	// Statemachine
	eStep					:E_ModbusRtuMaster_State;	// State
	eStepPrevious			:E_ModbusRtuMaster_State;	// State from previous scan
	eStatePrevious			:E_ModbusRtuMaster_State;	// Previous state
	nStepSecCount			:UDINT;						// Counts number of seconds without state transitions
	wStateSecOld			:WORD;						// Seconds value from NtTime from previous scan	
	eStepEntry				:BOOL;						// True in one scan when a new state is entered
	arrStateLog				:ARRAY[0..19] OF ST_ModbusRtuMaster_StateLogEntry; // Log that contains the last xx states
	
	// Modbus master
	fbModBusMaster			:ModbusRtuMaster_KL6x22B;	// Modbus master functions
	bReadExe				:BOOL;						// On rising edge reading is started
	bReadBusy				:BOOL;						// True while modbus master reads register on unit
	bReadError				:BOOL;						// True if read error occured
	eReadErrorID			:MODBUS_ERRORS;				// Modbus error ID
	nReadNoOfBytes			:UINT;						// Nunber of bytes read in read cycle

	// Units
	nUnitActive				:INT;						// Active unit in cyclic read
	nParamActive			:INT;						// Active parameter in cyclic read
END_VAR
VAR CONSTANT
	cNoOfUnitsMax			:INT:= 20;					// Maximum number of units for modbus master
END_VAR


// Initialization	
IF bInit THEN	
	bInit := FALSE;
END_IF

// Wait for reset
IF bCmdReset THEN
	bCmdReset := FALSE;
	bError := FALSE;
	nErrorUnit := 0;
	bReadExe := FALSE;
	eStep := E_ModbusRtuMaster_State.eIdle;	
END_IF

// Update fb for modbus communication
IF eStep >= E_ModbusRtuMaster_State.eReadPre AND eStep <= E_ModbusRtuMaster_State.eReadPost THEN
	fbModbusMaster.ReadRegs(
		UnitID:= pUnit^[nUnitActive].nAddr, 
		Quantity:= pUnit^[nUnitActive].aParam[nParamActive].nQuantity, 
		MBAddr:= (pUnit^[nUnitActive].aParam[nParamActive].nMemAddr*10)-1, 
		cbLength:= pUnit^[nUnitActive].aParam[nParamActive].nQuantity*2, 
		pMemoryAddr:= ADR(pUnit^[nUnitActive].aParam[nParamActive].aDataStorage), 
		Execute:= bReadExe, 
		Timeout:= T#2S, 
		BUSY=> bReadBusy, 
		Error=> bReadError, 
		ErrorId=> eReadErrorID, 
		cbRead=> nReadNoOfBytes);	
END_IF

	
// State machine
//----------------------------------------
// Check for new state entry
IF eStep <> eStepPrevious THEN
	// New state, Set entry flag
	eStepEntry := TRUE;
	eStatePrevious := eStepPrevious;
ELSE
	// Same state as last scan, remove entry flag
	eStepEntry := FALSE;
END_IF
// Update state log
A_StateLog();
// Reset "old" state to present value
eStepPrevious := eStep;
	

CASE eStep OF
E_ModbusRtuMaster_State.eReset:
	eStep := E_ModbusRtuMaster_State.eIdle;	


E_ModbusRtuMaster_State.eIdle:
	// Entry
	IF eStepEntry THEN
		A_ResetAllCmd();
		bBusy 	:= FALSE;
		bError	:= FALSE;
		bReadExe := FALSE;
	END_IF
	// Wait for command
	IF bCmdCyclicRead THEN
		bBusy	 := TRUE;
		bReadExe := FALSE;
		bCmdCyclicRead := FALSE;
		nUnitActive := 1;
		nParamActive := 1;
		eStep := E_ModbusRtuMaster_State.eReadPre;
	END_IF
		
	
E_ModbusRtuMaster_State.eReadPre:
	// Send request for reading of hold register
	bReadExe := TRUE;
	//IF bReadBusy THEN
		eStep := E_ModbusRtuMaster_State.eReadPost;
	//END_IF	 
	
	
E_ModbusRtuMaster_State.eReadPost:
	// Wait for answer back
	IF NOT bReadBusy THEN
		IF NOT bReadError THEN
			// Successfull read
			nReadCount := nReadCount + 1;
			// Convert return data to value
			IF pUnit^[nUnitActive].aParam[nParamActive].eDataType = E_Modbus_DataType.eInt16 THEN
				nValueTempInt16 := FUN_ConvTwoByteToInt16(
									nValue1:= pUnit^[nUnitActive].aParam[nParamActive].aDataStorage[1],
									nValue2:= pUnit^[nUnitActive].aParam[nParamActive].aDataStorage[2]);
				pUnit^[nUnitActive].aParam[nParamActive].aDataValue := INT_TO_REAL(nValueTempInt16) * pUnit^[nUnitActive].aParam[nParamActive].fConvFactor;				
			ELSIF pUnit^[nUnitActive].aParam[nParamActive].eDataType = E_Modbus_DataType.eInt32 THEN
				nValueTempInt32 := FUN_ConvFourByteToInt32(
									nValue1:= pUnit^[nUnitActive].aParam[nParamActive].aDataStorage[3],
									nValue2:= pUnit^[nUnitActive].aParam[nParamActive].aDataStorage[4],
									nValue3:= pUnit^[nUnitActive].aParam[nParamActive].aDataStorage[1],
									nValue4:= pUnit^[nUnitActive].aParam[nParamActive].aDataStorage[2]);
				pUnit^[nUnitActive].aParam[nParamActive].aDataValue := DINT_TO_REAL(nValueTempInt32) * pUnit^[nUnitActive].aParam[nParamActive].fConvFactor; 
			END_IF
			// Determine next step
			IF NOT bCmdStop THEN
				// Update setting to next parameter (and unit if this was the last parameter)
				nParamActive := nParamActive + 1;
				IF nParamActive > nNoOfParam THEN
					// All parameters read from unit. Change to next unit
					nParamActive := 1;
					IF nUnitActive >= nNoOfUnits THEN
						// Loop back to first unit in array
						nUnitActive := 1;
					ELSE
						// Take next unit in array
						nUnitActive := nUnitActive + 1;
					END_IF		
				END_IF
				// Go back and start reading the next parameter
				bReadExe := FALSE;
				eStep := E_ModbusRtuMaster_State.eReadPre;
			ELSE
				// Stop cyclic reading of hold registers
				eStep := E_ModbusRtuMaster_State.eIdle;
			END_IF
		ELSE
			// Error occured
			eStep := E_ModbusRtuMaster_State.eError;	
		END_IF	
	END_IF

	
E_ModbusRtuMaster_State.eError:
	// Entry
	IF eStepEntry THEN
		A_ResetAllCmd();
		bBusy := FALSE;
		IF nErrorUnit = 0 THEN
			bError := TRUE;	 
			nErrorUnit := nUnitActive;
		END_IF
	END_IF
	
	// Go back and try next unit
	IF nUnitActive >= nNoOfUnits THEN
		// Loop back to first unit in array
		nUnitActive := 1;
	ELSE
		// Take next unit in array
		nUnitActive := nUnitActive + 1;
	END_IF
	// Go back and start reading the next parameter
	bReadExe := FALSE;
	eStep := E_ModbusRtuMaster_State.eReadPre;
	
	(*
	// Wait for reset
	IF bCmdReset THEN
		bCmdReset := FALSE;
		eStep := E_ModbusRtuMaster_State.eIdle;	
	END_IF
	*)
END_CASE

ACTION A_ResetAllCmd:
// Reset all commands
bCmdCyclicRead := FALSE;
bCmdStop  := FALSE;
bCmdReset := FALSE;
END_ACTION

ACTION A_StateLog:
// Action: State log
//---------------------------------------------------------------
// The code below implements a simple state log in RAM. The purpose of the log
// is to give the developer a state history when debugging.

// Seconds counter
//-----------------------------------------------
IF wStateSecOld <> GVL_System.stNtTime.wSecond THEN
	// New second => Update counter
	IF nStepSecCount >= 4294967294 THEN
		nStepSecCount := 0;
	END_IF
	nStepSecCount := nStepSecCount + 1;
END_IF  
wStateSecOld := GVL_System.stNtTime.wSecond;

// Update time in active state
//-----------------------------------------------
arrStateLog[0].iSecCount := nStepSecCount;

// Update Stringer state log
//-----------------------------------------------
IF 	(eStep <> eStepPrevious) THEN
	// New state transition has occured => make new entry in the state log
	// Start with shift in log (FIFO)
	MEMMOVE(
		destAddr:= ADR(arrStateLog[1]), 
		srcAddr:= ADR(arrStateLog[0]), 
		n:= (SIZEOF(arrStateLog) - SIZEOF(arrStateLog[0]))); 
		
	// Add new entry to start of log
	arrStateLog[0].eStep 		:= eStep; 
	arrStateLog[0].sTimeEntry 	:= FUN_GetTimestamp(GVL_System.stNtTime);
	arrStateLog[0].iSecCount 	:= 0;
	
	// Reset seconds counter
	nStepSecCount := 0;
END_IF
END_ACTION

METHOD M_CmdCyclicRead : BOOL
VAR_INPUT
END_VAR

// Check if it is a valid command
IF eStep = E_ModbusRtuMaster_State.eIdle THEN
	// Valid command
	bCmdCyclicRead := TRUE;
END_IF

// Return result for acceptance of command
IF bCmdCyclicRead THEN
	M_CmdCyclicRead := TRUE;
ELSE
	M_CmdCyclicRead := FALSE;
END_IF
END_METHOD

METHOD M_CmdReset : BOOL
VAR_INPUT
END_VAR

// Check if it is a valid command
IF eStep = E_ModbusRtuMaster_State.eError THEN
	// Valid command
	bCmdReset := TRUE;
END_IF

// Return result for acceptance of command
IF bCmdReset THEN
	M_CmdReset := TRUE;
ELSE
	M_CmdReset := FALSE;
END_IF
END_METHOD

METHOD M_CmdStop : BOOL
VAR_INPUT
END_VAR

// Check if it is a valid command
IF eStep > E_ModbusRtuMaster_State.eIdle AND eStep < E_ModbusRtuMaster_State.eError THEN
	// Valid command
	bCmdStop := TRUE;
END_IF

// Return result for acceptance of command
IF bCmdStop THEN
	M_CmdStop := TRUE;
ELSE
	M_CmdStop := FALSE;
END_IF
END_METHOD

END_FUNCTION_BLOCK

// ---- POUs/00_BuildingBlocks/StringFunctions/FUN_GetTimestamp.TcPOU
FUNCTION FUN_GetTimestamp : STRING
VAR_INPUT
	stNtTime		:TIMESTRUCT;
END_VAR
VAR
	sTimestamp		:STRING;
END_VAR

// Add data
sTimeStamp := FUN_GetDate(stNtTime);

// Add time
sTimestamp := CONCAT(sTimeStamp, ' ');
sTimestamp := CONCAT(sTimeStamp, FUN_GetTime(stNtTime));

// Return time stamp
FUN_GetTimestamp := sTimestamp;

END_FUNCTION

// ---- POUs/00_BuildingBlocks/StringFunctions/FUN_GetDate.TcPOU
FUNCTION FUN_GetDate : STRING
VAR_INPUT
	stNtTime		:TIMESTRUCT;
END_VAR
VAR
	sDate			:STRING;
END_VAR

// Initialize string
sDate := '';

// Add year to string
sDate := UINT_TO_STRING(stNtTime.wYear);
sDate := CONCAT(sDate,'-');

// Add month to string
IF stNtTime.wMonth < 10 THEN
	sDate := CONCAT(sDate,'0');
END_IF
sDate := CONCAT(sDate,UINT_TO_STRING(stNtTime.wMonth));
sDate := CONCAT(sDate,'-');

// Add day to string
IF stNtTime.wDay < 10 THEN
	sDate := CONCAT(sDate, '0');
END_IF
sDate := CONCAT(sDate,UINT_TO_STRING(stNtTime.wDay));

// Return result
FUN_GetDate := sDate;

END_FUNCTION

// ---- POUs/00_BuildingBlocks/StringFunctions/FUN_GetTime.TcPOU
FUNCTION FUN_GetTime : STRING
VAR_INPUT
	stNtTime		:TIMESTRUCT;
END_VAR
VAR
	sTimestamp		:STRING;
END_VAR

// Add hour to timestamp
sTimestamp := '';
IF stNtTime.wHour < 10 THEN
	sTimestamp := CONCAT(sTimestamp,CONCAT('0', UINT_TO_STRING(stNtTime.wHour)));
ELSE
	sTimestamp := CONCAT(sTimestamp,UINT_TO_STRING(stNtTime.wHour));
END_IF

// Add min to timestamp
sTimestamp := CONCAT(sTimestamp, ':');
IF stNtTime.wMinute < 10 THEN
	sTimestamp := CONCAT(sTimestamp,CONCAT('0', UINT_TO_STRING(stNtTime.wMinute)));
ELSE
	sTimestamp := CONCAT(sTimestamp,UINT_TO_STRING(stNtTime.wMinute));
END_IF
sTimestamp := CONCAT(sTimestamp, ':');

// Add sec to timestamp
IF stNtTime.wSecond < 10 THEN
	sTimestamp := CONCAT(sTimestamp,CONCAT('0', UINT_TO_STRING(stNtTime.wSecond)));
ELSE
	sTimestamp := CONCAT(sTimestamp,UINT_TO_STRING(stNtTime.wSecond));
END_IF

// Return time
FUN_GetTime := sTimestamp;

END_FUNCTION

// ---- POUs/00_BuildingBlocks/Modbus/FB_ModbusRtuMaster_20220719_1144.TcPOU
// FB_ModbusMaster
//------------------------------------------------------ 
// This FB must be called in a 2 ms task and in every scan
// Test with Danfoss FC301 shows that up to approximately 46 registers can be read pr. sec.
// Test was done with baud 115200. 
FUNCTION_BLOCK FB_ModbusRtuMaster_20220719_1144
VAR_INPUT
	pUnit					:POINTER TO ARRAY[1..cNoOfUnitsMax] OF ST_Modbus_Unit;
	nNoOfUnits				:INT;			// Number of modbus units. Maximum value is 20.					
	nNoOfParam				:INT;			// Number of modbus parameters to be read from unit. Maximum value is determined by ST_Modbus_Unit. 
END_VAR
VAR_OUTPUT
	bBusy					:BOOL;			// True while command is beeing executed
	bError					:BOOL;			// True if an error occured during execution of a command
END_VAR
VAR
	// Commands
	bCmdCyclicRead			:BOOL;			// Command for cyclic reading of parameter registers
	bCmdStop				:BOOL;			// Command for stop
	bCmdReset				:BOOL;			// Command for reset of active errors
	
	// General	
	bInit					:BOOL := TRUE;	// True at the start of false scan, false otherwise
	nReadCount				:INT;			// Counts the number of succesfull read operations
	nValueTempInt16			:INT;			// Value used in conversion from byte data to actual data value
	nValueTempInt32			:DINT;			// Value used in conversion from byte data to actual data value
	
	// Statemachine
	eStep					:E_ModbusRtuMaster_State;	// State
	eStepPrevious				:E_ModbusRtuMaster_State;	// State from previous scan
	eStatePrevious			:E_ModbusRtuMaster_State;	// Previous state
	nStepSecCount			:UDINT;						// Counts number of seconds without state transitions
	wStateSecOld			:WORD;						// Seconds value from NtTime from previous scan	
	eStepEntry				:BOOL;						// True in one scan when a new state is entered
	arrStateLog				:ARRAY[0..19] OF ST_ModbusRtuMaster_StateLogEntry; // Log that contains the last xx states
	
	// Modbus master
	fbModBusMaster			:ModbusRtuMaster_KL6x22B;	// Modbus master functions
	bReadExe				:BOOL;						// On rising edge reading is started
	bReadBusy				:BOOL;						// True while modbus master reads register on unit
	bReadError				:BOOL;						// True if read error occured
	eReadErrorID			:MODBUS_ERRORS;				// Modbus error ID
	nReadNoOfBytes			:UINT;						// Nunber of bytes read in read cycle

	// Units
	nUnitActive				:INT;						// Active unit in cyclic read
	nParamActive			:INT;						// Active parameter in cyclic read
END_VAR
VAR CONSTANT
	cNoOfUnitsMax			:INT:= 20;					// Maximum number of units for modbus master
END_VAR


// Initialization	
IF bInit THEN	
	bInit := FALSE;
END_IF


// Update fb for modbus communication
IF eStep >= E_ModbusRtuMaster_State.eReadPre AND eStep <= E_ModbusRtuMaster_State.eReadPost THEN
	fbModbusMaster.ReadRegs(
		UnitID:= pUnit^[nUnitActive].nAddr, 
		Quantity:= pUnit^[nUnitActive].aParam[nParamActive].nQuantity, 
		MBAddr:= (pUnit^[nUnitActive].aParam[nParamActive].nMemAddr*10)-1, 
		cbLength:= pUnit^[nUnitActive].aParam[nParamActive].nQuantity*2, 
		pMemoryAddr:= ADR(pUnit^[nUnitActive].aParam[nParamActive].aDataStorage), 
		Execute:= bReadExe, 
		Timeout:= T#2S, 
		BUSY=> bReadBusy, 
		Error=> bReadError, 
		ErrorId=> eReadErrorID, 
		cbRead=> nReadNoOfBytes);	
END_IF

	
// State machine
//----------------------------------------
// Check for new state entry
IF eStep <> eStepPrevious THEN
	// New state, Set entry flag
	eStepEntry := TRUE;
	eStatePrevious := eStepPrevious;
ELSE
	// Same state as last scan, remove entry flag
	eStepEntry := FALSE;
END_IF
// Update state log
A_StateLog();
// Reset "old" state to present value
eStepPrevious := eStep;
	

CASE eStep OF
E_ModbusRtuMaster_State.eReset:
	eStep := E_ModbusRtuMaster_State.eIdle;	


E_ModbusRtuMaster_State.eIdle:
	// Entry
	IF eStepEntry THEN
		A_ResetAllCmd();
		bBusy 	:= FALSE;
		bError	:= FALSE;
		bReadExe := FALSE;
	END_IF
	// Wait for command
	IF bCmdCyclicRead THEN
		bBusy	 := TRUE;
		bReadExe := FALSE;
		bCmdCyclicRead := FALSE;
		nUnitActive := 1;
		nParamActive := 1;
		eStep := E_ModbusRtuMaster_State.eReadPre;
	END_IF
		
	
E_ModbusRtuMaster_State.eReadPre:
	// Send request for reading of hold register
	bReadExe := TRUE;
	//IF bReadBusy THEN
		eStep := E_ModbusRtuMaster_State.eReadPost;
	//END_IF	 
	
	
E_ModbusRtuMaster_State.eReadPost:
	// Wait for answer back
	IF NOT bReadBusy THEN
		IF NOT bReadError THEN
			// Successfull read
			nReadCount := nReadCount + 1;
			// Convert return data to value
			IF pUnit^[nUnitActive].aParam[nParamActive].eDataType = E_Modbus_DataType.eInt16 THEN
				nValueTempInt16 := FUN_ConvTwoByteToInt16(
									nValue1:= pUnit^[nUnitActive].aParam[nParamActive].aDataStorage[1],
									nValue2:= pUnit^[nUnitActive].aParam[nParamActive].aDataStorage[2]);
				pUnit^[nUnitActive].aParam[nParamActive].aDataValue := INT_TO_REAL(nValueTempInt16) * pUnit^[nUnitActive].aParam[nParamActive].fConvFactor;				
			ELSIF pUnit^[nUnitActive].aParam[nParamActive].eDataType = E_Modbus_DataType.eInt32 THEN
				nValueTempInt32 := FUN_ConvFourByteToInt32(
									nValue1:= pUnit^[nUnitActive].aParam[nParamActive].aDataStorage[3],
									nValue2:= pUnit^[nUnitActive].aParam[nParamActive].aDataStorage[4],
									nValue3:= pUnit^[nUnitActive].aParam[nParamActive].aDataStorage[1],
									nValue4:= pUnit^[nUnitActive].aParam[nParamActive].aDataStorage[2]);
				pUnit^[nUnitActive].aParam[nParamActive].aDataValue := DINT_TO_REAL(nValueTempInt32) * pUnit^[nUnitActive].aParam[nParamActive].fConvFactor; 
			END_IF
			// Determine next step
			IF NOT bCmdStop THEN
				// Update setting to next parameter (and unit if this was the last parameter)
				nParamActive := nParamActive + 1;
				IF nParamActive > nNoOfParam THEN
					// All parameters read from unit. Change to next unit
					nParamActive := 1;
					IF nUnitActive >= nNoOfUnits THEN
						// Loop back to first unit in array
						nUnitActive := 1;
					ELSE
						// Take next unit in array
						nUnitActive := nUnitActive + 1;
					END_IF		
				END_IF
				// Go back and start reading the next parameter
				bReadExe := FALSE;
				eStep := E_ModbusRtuMaster_State.eReadPre;
			ELSE
				// Stop cyclic reading of hold registers
				eStep := E_ModbusRtuMaster_State.eIdle;
			END_IF
		ELSE
			// Error occured
			eStep := E_ModbusRtuMaster_State.eError;	
		END_IF	
	END_IF

	
E_ModbusRtuMaster_State.eError:
	// Entry
	IF eStepEntry THEN
		A_ResetAllCmd();
		bBusy := FALSE;
		bError := TRUE;	
	END_IF
	// Wait for reset
	IF bCmdReset THEN
		bCmdReset := FALSE;
		eStep := E_ModbusRtuMaster_State.eIdle;	
	END_IF
END_CASE

ACTION A_ResetAllCmd:
// Reset all commands
bCmdCyclicRead := FALSE;
bCmdStop  := FALSE;
bCmdReset := FALSE;
END_ACTION

ACTION A_StateLog:
// Action: State log
//---------------------------------------------------------------
// The code below implements a simple state log in RAM. The purpose of the log
// is to give the developer a state history when debugging.

// Seconds counter
//-----------------------------------------------
IF wStateSecOld <> GVL_System.stNtTime.wSecond THEN
	// New second => Update counter
	IF nStepSecCount >= 4294967294 THEN
		nStepSecCount := 0;
	END_IF
	nStepSecCount := nStepSecCount + 1;
END_IF  
wStateSecOld := GVL_System.stNtTime.wSecond;

// Update time in active state
//-----------------------------------------------
arrStateLog[0].iSecCount := nStepSecCount;

// Update Stringer state log
//-----------------------------------------------
IF 	(eStep <> eStepPrevious) THEN
	// New state transition has occured => make new entry in the state log
	// Start with shift in log (FIFO)
	MEMMOVE(
		destAddr:= ADR(arrStateLog[1]), 
		srcAddr:= ADR(arrStateLog[0]), 
		n:= (SIZEOF(arrStateLog) - SIZEOF(arrStateLog[0]))); 
		
	// Add new entry to start of log
	arrStateLog[0].eStep 		:= eStep; 
	arrStateLog[0].sTimeEntry 	:= FUN_GetTimestamp(GVL_System.stNtTime);
	arrStateLog[0].iSecCount 	:= 0;
	
	// Reset seconds counter
	nStepSecCount := 0;
END_IF
END_ACTION

METHOD M_CmdCyclicRead : BOOL
VAR_INPUT
END_VAR

// Check if it is a valid command
IF eStep = E_ModbusRtuMaster_State.eIdle THEN
	// Valid command
	bCmdCyclicRead := TRUE;
END_IF

// Return result for acceptance of command
IF bCmdCyclicRead THEN
	M_CmdCyclicRead := TRUE;
ELSE
	M_CmdCyclicRead := FALSE;
END_IF
END_METHOD

METHOD M_CmdReset : BOOL
VAR_INPUT
END_VAR

// Check if it is a valid command
IF eStep = E_ModbusRtuMaster_State.eError THEN
	// Valid command
	bCmdReset := TRUE;
END_IF

// Return result for acceptance of command
IF bCmdReset THEN
	M_CmdReset := TRUE;
ELSE
	M_CmdReset := FALSE;
END_IF
END_METHOD

METHOD M_CmdStop : BOOL
VAR_INPUT
END_VAR

// Check if it is a valid command
IF eStep > E_ModbusRtuMaster_State.eIdle AND eStep < E_ModbusRtuMaster_State.eError THEN
	// Valid command
	bCmdStop := TRUE;
END_IF

// Return result for acceptance of command
IF bCmdStop THEN
	M_CmdStop := TRUE;
ELSE
	M_CmdStop := FALSE;
END_IF
END_METHOD

END_FUNCTION_BLOCK

// ---- POUs/00_BuildingBlocks/Modbus/PRG_ModbusTest.TcPOU
PROGRAM PRG_ModbusTest
VAR
	// General	
	bInit					:BOOL := TRUE;
	nForIndex				:INT;
	
	bTestCyclicRead			:BOOL;
	bTestStop				:BOOL;
	bTestReset				:BOOL;
	
	// Modbus
	fbModbus				:FB_ModbusRtuMaster;
	fbModbusBusy			:BOOL;
	fbModbusError			:BOOL;
	
	// Frequency inverters
	aVFD					:ARRAY[1..cNoOfUnits] OF ST_Modbus_Unit; 	
END_VAR
VAR CONSTANT
	cNoOfUnits				:INT:= 2;
	cNoOfParam				:INT:= 4;
END_VAR


// Initialization
//-------------------------------------------	
IF bInit THEN	
	// VFD address 
	aVFD[1].nAddr := 2;
	aVFD[2].nAddr := 3;
	// Parameters to be read in each VFD
	FOR nForIndex := 1 TO cNoOfUnits BY 1 DO
		aVFD[nForIndex].aParam[1].nMemAddr 		:= 1610;	 				 // [W] Power (Value back is in W and not kW)
		aVFD[nForIndex].aParam[1].nQuantity 	:= 4;						 // Bytes
		aVFD[nForIndex].aParam[1].fConvFactor 	:= 10.0; 				     // Conversion index 1 => Conversion factor 10
		aVFD[nForIndex].aParam[1].eDataType 	:= E_Modbus_DataType.eInt32; // Int32
		
		aVFD[nForIndex].aParam[2].nMemAddr 		:= 1612;					// [V] Motor voltage
		aVFD[nForIndex].aParam[2].nQuantity 	:= 2;						// Bytes -> 2 bytes
		aVFD[nForIndex].aParam[2].fConvFactor 	:= 0.1; 					// Conversion index -1 => Conversion factor 0.1
		aVFD[nForIndex].aParam[2].eDataType 	:= E_Modbus_DataType.eInt16;// Int16 
		
		aVFD[nForIndex].aParam[3].nMemAddr 		:= 1613;					// [Hz] Frequency
		aVFD[nForIndex].aParam[3].nQuantity 	:= 2;						// Bytes
		aVFD[nForIndex].aParam[3].fConvFactor 	:= 0.1; 					// Conversion index -1 => Conversion factor 0.1
		aVFD[nForIndex].aParam[3].eDataType 	:= E_Modbus_DataType.eInt16;// Int16 
		
		aVFD[nForIndex].aParam[4].nMemAddr 		:= 1614;					// [A] Motor current 
		aVFD[nForIndex].aParam[4].nQuantity 	:= 4;						// Bytes
		aVFD[nForIndex].aParam[4].fConvFactor 	:= 0.01;				 	// Conversion index -2 => Conversion factor 0.01
		aVFD[nForIndex].aParam[4].eDataType 	:= E_Modbus_DataType.eInt32;// Int32
	END_FOR
	bInit := FALSE;
END_IF


// Update function block that handles modbus communication
//-------------------------------------------	
fbModbus(
	pUnit:= ADR(aVFD),
	nNoOfUnits := cNoOfUnits,
	nNoOfParam := cNoOfParam,
	bBusy => fbModbusBusy,
	bError => fbModbusError);

	
// Commands	
//-------------------------------------------		
// Test/Start cyclic read of data
IF bTestCyclicRead THEN
	fbModbus.M_CmdCyclicRead();
	bTestCyclicRead := FALSE;
END_IF

// Stop cyclic read of data
IF bTestStop THEN
	fbModbus.M_CmdStop();
	bTestStop := FALSE;
END_IF

// Reset of error
IF bTestReset THEN
	fbModbus.M_CmdReset();
	bTestReset := FALSE;
END_IF

	
// Results (Read outs)
//-------------------------------------
// VFD 1
//aVFD[1].aParam[1].aDataValue;		// [W] Power
//aVFD[1].aParam[2].aDataValue;		// [V] Motor voltage
//aVFD[1].aParam[3].aDataValue;		// [Hz] Frequency
//aVFD[1].aParam[4].aDataValue;		// [A] Motor current 

// VFD 2
//aVFD[2].aParam[1].aDataValue;		// [W] Power
//aVFD[2].aParam[2].aDataValue;		// [V] Motor voltage
//aVFD[2].aParam[3].aDataValue;		// [Hz] Frequency
//aVFD[2].aParam[4].aDataValue;		// [A] Motor current

END_PROGRAM

// ---- POUs/00_BuildingBlocks/PlcToPlcCom/FB_PlcAdsRead.TcPOU
//**************************************************************************
// FB_PlcAdsRead
// -------------------------------------------------------------------------
// This FB reads the content of a variable or struct from a remote PLC. The
// FB is usefull when data needs to be exchaged between two PLC's. The FB only
// reads the content from the other PLC, it does NOT write any variables. Hence
// the same FB will need to be implemented on other PLC, which then reads the
// commands/variables that needs to be sent.  
//
// Version
//		- V1.00.00	HHL, 21/08-2019
//**************************************************************************
FUNCTION_BLOCK FB_PlcAdsRead
VAR_INPUT
	sRemoteNetId 		:STRING; 			// Remote plc NetId
	uiRemoteAmsPort 	:UINT := 851; 		// Ams port 
	sSymbolName 		:STRING := '';		// Symbol name on remote PLC
	dwAddress 			:PVOID; 			// Variable address at local system. Name must be the same at remote
	udiLength 			:UDINT; 			// Variable length at local system. Name must be the same at remote
	tReadInterval 		:TIME := T#1S; 		// Read interval
	tReadTimeout 		:TIME := T#2S; 		// Read timeout
	
	bEnable 			:BOOL := TRUE; 		// Enable communication
	bStartRead			:BOOL;				// Force Start Read  Started
END_VAR
VAR_OUTPUT
	bLinkOk 			:BOOL; 				// Link to remote plc is ok
	bError 				:BOOL; 				// Connection error
	
	eErrorStep 			:E_PlcAdsReadStep; 	// Error step
	udiErrorId 			:UDINT; 			// Error id (ads)
END_VAR
VAR
	bEntry 				:BOOL;
	udiHandle 			:UDINT; 			// Handel
	sSymbolNameEdge 	:STRING;
	
	eStep, eStepEdge 	:E_PlcAdsReadStep;
	stHmi 				:ST_PlcAdsReadHmi; 	// Hmi data
	
	fbAdsRdWrt 			:ADSRDWRT;
	fbAdsRead 			:ADSREAD;
	fbInitRetry 		:TON; 				// Delay before retry
	fbReadInterval 		:TON; 				// Read interval timer
	osStartReadADS		:R_TRIG;			// os Start Read ADS Data
	// Force Start Read Started
	bForceStartRead: BOOL;
END_VAR

osStartReadADS(CLK:=bStartRead , Q=> );

IF osStartReadADS.Q THEN
	bForceStartRead:=TRUE;
END_IF

bEntry := eStepEdge<>eStep;
eStepEdge := eStep;


CASE eStep OF
	//-----------------------------
	// Init
	E_PlcAdsReadStep.eReset:	
		fbAdsRdWrt.WRTRD := FALSE;	
		fbAdsRead.READ := FALSE;
		
		bLinkOk := FALSE;
		bError := FALSE;
		udiErrorId := 0;
		eErrorStep := E_PlcAdsReadStep.eReset;

		eStep := E_PlcAdsReadStep.eGetRemoteInfo;	
	
	//-----------------------------
	// Get info (Index-Group/Offset)
	E_PlcAdsReadStep.eGetRemoteInfo:
		IF bEntry THEN
			fbAdsRdWrt.WRTRD := TRUE;
		END_IF
		
		IF fbAdsRdWrt.BUSY THEN
			//Read started
			eStep := E_PlcAdsReadStep.eWaitRemoteInfo;
		END_IF
	
	//-----------------------------
	// Wait for remote info
	E_PlcAdsReadStep.eWaitRemoteInfo:
		IF NOT fbAdsRdWrt.BUSY THEN
			IF NOT fbAdsRdWrt.ERR THEN
				//Get remote info ok
				sSymbolNameEdge := sSymbolName;
				IF bEnable OR bForceStartRead THEN
					eStep := E_PlcAdsReadStep.eRead;
					bForceStartRead:=FALSE;
				ELSE
					eStep := E_PlcAdsReadStep.eIdle;
				END_IF
			ELSE
				//Get remote info failed
				eErrorStep := eStep;
				udiErrorId := fbAdsRdWrt.ERRID;
				
				eStep := E_PlcAdsReadStep.eGetInfoError;
			END_IF
		END_IF
	
	//-----------------------------
	// Get info failed
	E_PlcAdsReadStep.eGetInfoError:		
		IF fbInitRetry.Q THEN
			//Retry
			eStep := E_PlcAdsReadStep.eReset;
		END_IF
		
	//-----------------------------
	// Idle
	E_PlcAdsReadStep.eIdle:		
		IF bEntry THEN
			fbAdsRead.READ := FALSE;
		END_IF
		
		IF bEnable OR bForceStartRead THEN
			IF FIND(STR1:=sSymbolName, STR2:=sSymbolNameEdge)=1 THEN
				//Symbol has'nt changed
				eStep := E_PlcAdsReadStep.eRead;
				bForceStartRead:=FALSE;
			ELSE
				eStep := E_PlcAdsReadStep.eReset;
			END_IF
			
		END_IF
	
	//-----------------------------
	// Read data
	E_PlcAdsReadStep.eRead:	
		IF bEntry THEN
			//Start read
			fbAdsRead.READ := TRUE;
			eErrorStep := E_PlcAdsReadStep.eIdle;
			udiErrorId := 0;
		END_IF
		
		IF fbAdsRead.BUSY THEN
			//Read started
			eStep := E_PlcAdsReadStep.eWaitReadDone;
		END_IF
	
	//-----------------------------
	// Wait read finished
	E_PlcAdsReadStep.eWaitReadDone:
		IF NOT fbAdsRead.BUSY THEN
			stHmi.udiS_ReadCount := stHmi.udiS_ReadCount + 1;
			IF NOT fbAdsRead.ERR THEN
				bLinkOk := TRUE;
				eStep := E_PlcAdsReadStep.eWaitBeforeNextRead;
			ELSE
				bLinkOk := FALSE;
				eStep := E_PlcAdsReadStep.eReadError;
			END_IF
		END_IF
	
	//-----------------------------	
	// Wait before next read
	E_PlcAdsReadStep.eWaitBeforeNextRead:
		IF bEntry THEN
			fbAdsRead.READ := FALSE;
		END_IF
		
		IF fbReadInterval.Q THEN
			eStep := E_PlcAdsReadStep.eRead;
		END_IF
	
	//-----------------------------
	// Read failed
	E_PlcAdsReadStep.eReadError:
		IF bEntry THEN
			//Get remote info failed
			eErrorStep := eStep;
			udiErrorId := fbAdsRead.ERRID;
			stHmi.udiS_ReadErrors := stHmi.udiS_ReadErrors + 1;
		END_IF
		
		IF fbInitRetry.Q THEN
			// Try to init
			eStep := E_PlcAdsReadStep.eReset;
		END_IF
ELSE
	eStep := E_PlcAdsReadStep.eReset;
END_CASE

//Timers
fbReadInterval(IN:=NOT fbReadInterval.Q, PT:=tReadInterval);
IF fbReadInterval.Q AND (eStep=E_PlcAdsReadStep.eRead OR eStep=E_PlcAdsReadStep.eWaitReadDone) THEN
	//Read interval error
	stHmi.udiS_ReadIntervalErrors := stHmi.udiS_ReadIntervalErrors + 1;
END_IF
fbInitRetry(IN:=eStep=E_PlcAdsReadStep.eGetInfoError OR eStep=E_PlcAdsReadStep.eReadError, PT:=T#10S);

//Init
IF stHmi.bC_Init THEN
	eStep := E_PlcAdsReadStep.eReset;
	stHmi.bC_Init := FALSE;
END_IF

//Calls
fbAdsRdWrt(
	NETID:=sRemoteNetId, 
	PORT:=uiRemoteAmsPort, 
	IDXGRP:=16#F003, //GET_SYMHANDLE_BYNAME
	IDXOFFS:= 16#0000, 
	WRITELEN:= SIZEOF(sSymbolName),
	READLEN:= SIZEOF(udiHandle), 
	SRCADDR:= ADR(sSymbolName),
	DESTADDR:= ADR(udiHandle), 
	WRTRD:= , 
	TMOUT:=DEFAULT_ADS_TIMEOUT, 
	BUSY=> , 
	ERR=> , 
	ERRID=> );

fbAdsRead(
	NETID:= sRemoteNetId,
	PORT:= uiRemoteAmsPort,
	IDXGRP:= 16#F005, // READ_/WRITE_SYMVAL_BYHANDLE
	IDXOFFS:= udiHandle,
	LEN:= udiLength,
	DESTADDR:= dwAddress,
	READ:= ,
	TMOUT:= tReadTimeout,
	BUSY=> ,
	ERR=> ,
	ERRID=> );
	
A_HMI();

ACTION A_HMI:
stHmi.sRemoteId := sRemoteNetId;
stHmi.sRemoteSymbol := sSymbolName;
stHmi.bS_Enable := bEnable;
stHmi.bS_LinkOk := bLinkOk;
stHmi.bS_Error := bError;
stHmi.eS_Step := eStep;
stHmi.eS_ErrorStep := eErrorStep;
stHmi.udiS_ErrorId := udiErrorId;
END_ACTION

END_FUNCTION_BLOCK

// ---- POUs/00_BuildingBlocks/PlcToPlcCom/PRG_PlcAdsRead_Example.TcPOU
PROGRAM PRG_PlcAdsRead_Example
VAR
	fbPlcToPlc		:FB_PlcAdsRead;			// Function block that reads a struct from a remote PLC
	stDataToPlc		:ST_ComTest;			// Data to be read from remote PLC (same type of struct must be implemented on remote PLC)
END_VAR


// Call FB that reads struct on remote PLC
fbPlcToPlc(
	sRemoteNetId:= '192.168.1.3.1.1', 			// AMS net id on remote PLC
	uiRemoteAmsPort:= 851, 
	sSymbolName:= 'GVL_Interface.stData', 		// Symbol name on remote PLC
	dwAddress:= ADR(stDataToPlc), 				// Addres where data from remote PLC must be stored
	udiLength:= SIZEOF(stDataToPlc), 			// Size of data that is rad
	tReadInterval:= T#1S, 
	tReadTimeout:= T#2S, 
	bEnable:= , 
	bStartRead:= , 
	bLinkOk=> , 
	bError=> , 
	eErrorStep=> , 
	udiErrorId=> );

END_PROGRAM

// ---- POUs/00_BuildingBlocks/StringFunctions/FB_SeperateFileAndPathName.TcPOU
FUNCTION_BLOCK FB_SeperateFileAndPathName
VAR_INPUT
	sPathAndFileName	:STRING(255);	// String with path and file name
END_VAR
VAR_OUTPUT
	sFileName			:STRING(80);	// String with file name
	sPathName			:STRING(175);	// String with path name
	bError				:BOOL;			// True if error occured during determination of file and path name
END_VAR
VAR
	iLength				:INT;			// Length of string that is examined
	iPos				:INT;			// Charactor position used to seperate file name from string
	iSize				:INT;			// Size of a string
	sTemp				:STRING;		// Temporary string
	iForIndex			:INT;			// Index used in for-loops
	bSeperatorFound		:BOOL;			// True if charator for folder seperator was found in input string
END_VAR


// Initialize flag for seperator found
bSeperatorFound := FALSE;

// Search through string and find the last "\" charactor
iLength := LEN(sPathAndFileName);
FOR iForIndex := 1 TO iLength BY 1 DO
	IF MID(sPathAndFileName,1,iForIndex) = '\' THEN
		iPos := iForIndex;
		bSeperatorFound := TRUE;
	END_IF
END_FOR

IF bSeperatorFound THEN
	// Set file name
	iSize := iLength - iPos;
	sFileName := RIGHT(sPathAndFileName,iSize);
	
	// Set path name
	sPathName := LEFT(sPathAndFileName,iPos);
	
	// Reset error flag
	bError := FALSE;
ELSE
	// Set error flag
	bError := TRUE;
END_IF

END_FUNCTION_BLOCK

// ---- POUs/00_BuildingBlocks/StringFunctions/FUN_AddValuleToString.TcPOU
FUNCTION FUN_AddValuleToString : STRING(490)
VAR_INPUT
	sString		:STRING(490);	// String where value is to be added
	rValue		:LREAL;			// Value to be added to string
	iNoOfDec	:INT;			// Number of decimals to be presented in the string
END_VAR
VAR
	sSeperator	:STRING(80);	// Seperator
	sValue		:STRING(80);	// String version of value
END_VAR


// Create string for value
sValue := FUN_RealToString(rValue:= rValue, iNoOfDec:= iNoOfDec);

// Replace "." character with "," character (special Elvstrøm request)
sValue := FUN_ReplaceDotWithComma(sStringIn:= sValue);

// Add seperator to string
sSeperator := ';';
CONCAT2(pSrcString1:= ADR(sString), pSrcString2:= ADR(sSeperator), pDstString:= ADR(sString), nDstSize:= 490);

// Add value to string
CONCAT2(pSrcString1:= ADR(sString), pSrcString2:= ADR(sValue), pDstString:= ADR(sString), nDstSize:= 490);

// Return string
FUN_AddValuleToString := sString;

END_FUNCTION

// ---- POUs/00_BuildingBlocks/StringFunctions/FUN_RealToString.TcPOU
FUNCTION FUN_RealToString : STRING
VAR_INPUT
	rValue		:LREAL;			// Input value to be converted into a string
	iNoOfDec	:INT;			// Number of decimals to be presented in the string
END_VAR
VAR
	bNegative	:BOOL;			// True if value is negative
	i			:INT;			// Index used in for-loop
	iPos		:INT;			// Variable used to find position in string
	iPos2		:INT;			// Variable used to find position in string
	rTemp		:LREAL;			// Temporary value
	sTemp		:STRING;		// String version of rTemp
END_VAR

(* Set flag for negative number *)
(* If negative then multiply with -1. Function will then make conversion and insert - sign at the end *)
IF rValue < 0 THEN
	bNegative := TRUE;
	rValue := rValue * -1;
ELSE
	bNegative := FALSE;
END_IF


(* Multiply input value so that decimal part can be handleded without e- syntax *)
rTemp:= rValue;
FOR i:= 1 TO iNoOfDec DO
	rTemp := rTemp * 10;
END_FOR

IF rValue >= 1.0 THEN
	(* Input value does not contain the e- character. Normal conversion is possible *)
	sTemp := LREAL_TO_STRING(rTemp);

	(* Remove round off error *)
	IF MID(sTemp, 1, FIND(sTemp, '.')+1) = '9' THEN
		rTemp := rTemp + 0.1;
		FOR i:= 1 TO iNoOfDec DO
			rTemp := rTemp / 10;
		END_FOR
		sTemp := LREAL_TO_STRING(rTemp);
	ELSE
		sTemp := LREAL_TO_STRING(rValue);
	END_IF

	(* Examine length of decimal part of sTemp, and insert zeroes if needed. *)
	iPos := FIND(sTemp, '.');
	sTemp := LEFT(sTemp, iPos+iNoOfDec);
	iPos2 := LEN(sTemp);
	IF iPos2-iPos < iNoOfDec THEN
		(* Value is e.g. 1.0. Insert extra zero to get 1.0000 if number of decimals is 4 *)
		FOR i:= 1 TO (iNoOfDec- (iPos2-iPos)) DO
			sTemp := CONCAT(sTemp, '0');
		END_FOR
	END_IF
ELSE
	(* Input value does contain the e- character. Normal conversion is not possible *)
	sTemp := LREAL_TO_STRING(rTemp);

	(* Remove round off error *)
	IF MID(sTemp, 1, FIND(sTemp, '.')+1) = '9' THEN
		rTemp := rTemp + 0.1;
		sTemp := LREAL_TO_STRING(rTemp);
	END_IF

	IF rTemp > 1.0 THEN
		(* Value is greater than least significant decimal *)
		iPos := FIND(sTemp, '.');
		sTemp := DELETE(sTemp,1,iPos);
		FOR i:= 1 TO (iNoOfDec+2-iPos) DO
			sTemp := INSERT(sTemp, '0', 0);
		END_FOR
		sTemp := INSERT(sTemp, '.', 1);
		sTemp := LEFT(sTemp, iNoOfDec+2);

	ELSE
		(* Value is less than least significat decimal. Return all zero value *)
		sTemp := '0.0';
		FOR i :=1 TO iNoOfDec-1 DO
			sTemp := CONCAT(sTemp, '0');
		END_FOR
	END_IF
END_IF

(* Insert minus sign if input value was negative *)
IF bNegative THEN
	FUN_RealToString := CONCAT('-', sTemp);
ELSE
	FUN_RealToString := sTemp;
END_IF

END_FUNCTION

// ---- POUs/00_BuildingBlocks/StringFunctions/FUN_ReplaceDotWithComma.TcPOU
FUNCTION FUN_ReplaceDotWithComma: STRING(490)
VAR_INPUT
	sStringIn	:STRING(490);	// String where "." is used
END_VAR
VAR
	iLen		:INT;			// Number of characters in string
	iFindPos	:INT;			// Position in string where "." is found 
	iForIndex	:INT;			// Index used in for loops
	sStingOut	:STRING(490);	// String where "." has been replaced with ","		
END_VAR


// Initialize output string to input-string.
sStingOut := sStringIn;

// Get the length of the string
iLen := LEN(STR:=sStingOut);

IF iLen > 0 THEN
	// Go through string and replace all occurances of "."
	FOR iForIndex := 1 TO iLen BY 1 DO
		// Find "." in string
		iFindPos := FIND(STR1:= sStingOut, STR2:= '.');
		IF iFindPos > 0 THEN
			// Minimum one instance of "." is found. Replace this occurance.
			sStingOut := REPLACE(STR1:= sStingOut, STR2:= ',', L:= 1, P:=iFindPos);
		ELSE
			// All occurances have been found, terminate for-loop
			iForIndex := iLen + 1;
		END_IF
	END_FOR
ELSE
	// No charachters, output string is set equal to input
	;	
END_IF

// Return new string
FUN_ReplaceDotWithComma := sStingOut;

END_FUNCTION

// ---- POUs/00_BuildingBlocks/StringFunctions/FUN_GetDateWithoutSeperator.TcPOU
FUNCTION FUN_GetDateWithoutSeperator : STRING
VAR_INPUT
	stNtTime		:TIMESTRUCT;
END_VAR
VAR
	sDate			:STRING;
END_VAR

// Initialize string
sDate := '';

// Add year to string
sDate := UINT_TO_STRING(stNtTime.wYear);

// Add month to string
IF stNtTime.wMonth < 10 THEN
	sDate := CONCAT(sDate,'0');
END_IF
sDate := CONCAT(sDate,UINT_TO_STRING(stNtTime.wMonth));

// Add day to string
IF stNtTime.wDay < 10 THEN
	sDate := CONCAT(sDate, '0');
END_IF
sDate := CONCAT(sDate,UINT_TO_STRING(stNtTime.wDay));

// Return result
FUN_GetDateWithoutSeperator := sDate;

END_FUNCTION

// ---- POUs/00_BuildingBlocks/StringFunctions/FUN_GetDateWithUnderscore.TcPOU
FUNCTION FUN_GetDateWithUnderscore : STRING
VAR_INPUT
	stNtTime		:TIMESTRUCT;
END_VAR
VAR
	sDate			:STRING;
END_VAR

// Initialize string
sDate := '';

// Add year to string
sDate := UINT_TO_STRING(stNtTime.wYear);
sDate := CONCAT(sDate,'_');

// Add month to string
IF stNtTime.wMonth < 10 THEN
	sDate := CONCAT(sDate,'0');
END_IF
sDate := CONCAT(sDate,UINT_TO_STRING(stNtTime.wMonth));
sDate := CONCAT(sDate,'_');

// Add day to string
IF stNtTime.wDay < 10 THEN
	sDate := CONCAT(sDate, '0');
END_IF
sDate := CONCAT(sDate,UINT_TO_STRING(stNtTime.wDay));

// Return result
FUN_GetDateWithUnderscore := sDate;

END_FUNCTION

// ---- POUs/00_BuildingBlocks/StringFunctions/FUN_GetTimestampWithMs.TcPOU
FUNCTION FUN_GetTimestampWithMs : STRING
VAR_INPUT
	stNtTime		:TIMESTRUCT;				// Timestruct with present time
END_VAR
VAR
	sTimestamp		:STRING;					// String to contain timestamp text
	sMiliSec		:STRING;					// Miliseconds in timestamp
END_VAR

// Add data
//sTimeStamp := FUN_GetDate(stNtTime);

// Add time
//sTimestamp := CONCAT(sTimeStamp, ',');
//sTimestamp := CONCAT(sTimeStamp, FUN_GetTime(stNtTime));

// Get mili seconds value 
sMiliSec := '';
sMiliSec := UINT_TO_STRING(stNtTime.wMilliseconds);
IF stNtTime.wMilliseconds < 100 THEN
	sMiliSec := CONCAT(sMiliSec, '0');
	IF stNtTime.wMilliseconds < 10 THEN
		sMiliSec := CONCAT(sMiliSec, '0');
	END_IF
END_IF		

// Create and set timestamp
sTimeStamp := FUN_GetTimestamp(stNtTime);
sTimeStamp := CONCAT(STR1:= sTimeStamp, STR2:= '.'); 
sTimeStamp := CONCAT(STR1:= sTimeStamp, STR2:= sMiliSec); 
	
// Return time stamp
FUN_GetTimestampWithMs := sTimestamp;

END_FUNCTION

// ---- POUs/00_BuildingBlocks/StringFunctions/F_Replace.TcPOU
//------------------------------------------------------------------------------------------
//                                                                                        	
//***************************** Beckhoff TwinCAT Examples **********************************
//                                                                                        	
//************************************* WARNING ********************************************
// This program is only an example. If it is used as a control program in any real        	
// application, Beckhoff is not responsible for any malfunction, loss or damage           	
// which could arise by using this program!                                               	
//                                                                                        	
//*************************************  Program Info. *************************************
//                                                                                        	
// PLC program name:       	F_Replace2 (Function)               	                           	
// Software platform:      	TwinCat v3.1.4024.10				                          	
// Modified by:            	Per Søgaard Carlsen 			                                  	
// Email:					p.carlsen@beckhoff.com	                                  	
//                                                                                        	
// ======================================================================================== 
//         Version       Date                        Remarks                              	
// ======================================================================================== 
//         2.0           12 nov 2020                 First release of this example        	
// ======================================================================================== 
//                                                                                        	
//******************************* Aims OF this PLC PROGRAM *********************************
//                                                                                        	
// Compleate search and replace function in long strings						 			                             
//                                                                                        	
//-----------------------------------------------------------------------------------------
FUNCTION F_Replace : bool
VAR_INPUT
	sString : ANY_STRING; //String to search and replace
	sSearch : STRING(255); //Search in string
	sReplace : STRING(255); //Releace in string
END_VAR
VAR
	udiStartPos : UDINT; //Start position for found search result
	udiFindPos : UDINT; //Search start position in string
	bFoundOne : BOOL; //One ore more replace done
	bFoundThis : BOOL;
END_VAR

bFoundOne := FALSE; //Min one item replaced
udiFindPos := 0; //Search from position in string

REPEAT
	bFoundThis := FALSE;
	udiStartPos := udiFindPos;
	
	IF 	udiFindPos <= LEN2(pSTRING:= sString.pValue) THEN
		//Search
		udiFindPos := FIND2(pSrcString:= sString.pValue+udiStartPos, pFindString:= ADR(sSearch));
	ELSE
		//No match found
		udiFindPos := 0;
	END_IF
	
	IF udiFindPos <> 0 THEN
		//Replace item
		REPLACE2(
		pSrcString:= sString.pValue+udiStartPos, 
		pInsertString:= ADR(sReplace), 
		pDstString:= sString.pValue, 
		nDstSize:= TO_UDINT(sString.diSize)-udiStartPos, 
		nLen:= Tc2_Utilities.LEN2(ADR(sSearch)), 
		nPos:= udiFindPos);
		bFoundOne := TRUE;
		bFoundThis := TRUE;	
		
		udiFindPos := udiFindPos + TO_UDINT(Tc2_Standard.LEN(sReplace)); //Update search from position
		
		
	END_IF
	
	UNTIL NOT bFoundThis //Repeat until all item found and replaced
END_REPEAT

F_Replace := bFoundOne;

END_FUNCTION

// ---- POUs/01_TestUnit/TimeStampRegistry/FB_TimestampRegistryTest.TcPOU
FUNCTION_BLOCK FB_TimestampRegistryTest
VAR_INPUT
END_VAR
VAR_OUTPUT
END_VAR
VAR
END_VAR

END_FUNCTION_BLOCK

// ---- POUs/CSV_File/PRG_CSVRead.TcPOU
(* Reading of CSV file in text mode. None of the field value is containing any non-printing control characters like line feed, carriage return, quotation marks, semicolon... *)
PROGRAM PRG_CSVRead
VAR
	bRead			: BOOL := FALSE;(* Rising edge starts program execution *)
	sNetId			: T_AmsNetId := '';	(* TwinCAT system network address *)
	sFileName		: T_MaxString := 'C:\Temp\TextModeGen.csv';(* CSV source file path and name *)
	sCSVLine		: T_MaxString := '';(* Single CSV text line (row, record), we are using string as record buffer (your are able to see read fields)  *)
	sCSVField		: T_MaxString := '';(* Single CSV field value (column, record field) *)
	bBusy			: BOOL;
	bError			: BOOL;
	nErrId			: UDINT;
	nRow	 		: UDINT 	:= 0;(* Row number (record) *)
	nColumn			: UDINT 	:= 0;(* Column number (record field) *)
	hFile			: UINT		:= 0;(* File handle of the source file *)
	step			: DWORD 	:= 0;
	fbFileOpen		: FB_FileOpen;(* Opens file *)
	fbFileClose		: FB_FileClose;(* Closes file *)
	fbFileGets		: FB_FileGets;(* Reads one record (line) *)
	fbReader		: FB_CSVMemBufferReader;(* Helper function block used to parse CSV data bytes (single record line) *)

	database		: ARRAY[0..MAX_CSV_ROWS, 0..MAX_CSV_COLUMNS ] OF STRING(MAX_CSV_FIELD_LENGTH);(* Target PLC database *)
	nI				: INT;
	aItemEANRegistry: ARRAY[0..GVL_Constant.ITEM_ARRAY_SIZE] OF T_MaxString;
	aItemOnTime		: ARRAY[0..GVL_Constant.ITEM_ARRAY_SIZE] OF TIME;
	aItemOffTime	: ARRAY[0..GVL_Constant.ITEM_ARRAY_SIZE] OF TIME;
END_VAR

CASE step OF
	0:	(* Wait for rising edge at bRead variable *)
		IF bRead THEN
			bRead 	:= FALSE;
			bBusy 	:= TRUE;
			bError	:= FALSE;
			nErrId	:= 0;
			hFile	:= 0;
			nRow	:= 0;
			nColumn	:= 0;
			MEMSET( ADR( database ), 0, SIZEOF( database ) );
			step 		:= 1;
			
			FOR nI := 0 TO GVL_Constant.ITEM_ARRAY_SIZE DO
				aItemEANRegistry[nI] := database[nI, 0]; 
				aItemOnTime[nI] := STRING_TO_TIME(database[nI, 1]);  
				aItemOffTime[nI] := STRING_TO_TIME(database[nI, 2]); 
			END_FOR;
		END_IF

	1:	(* Open source file *)
		fbFileOpen(  bExecute := FALSE  );
		fbFileOpen( sNetId := sNetId, sPathName := sFileName, nMode := FOPEN_MODEREAD OR FOPEN_MODETEXT,(* Open file in TEXT mode! *)
					ePath := PATH_GENERIC, bExecute := TRUE );
		step := 2;

	2:(* Wait until open not busy *)
		fbFileOpen( bExecute := FALSE, bError => bError, nErrID => nErrID, hFile => hFile );
		IF NOT fbFileOpen.bBusy THEN
			IF NOT fbFileOpen.bError THEN
				step := 3;
			ELSE(* Error: file not found? *)
				step := 100;
			END_IF
		END_IF

	3:	(* Read single line (record) *)
		fbFileGets( bExecute := FALSE );
		fbFileGets( sNetId := sNetId, hFile := hFile, bExecute := TRUE );
		step := 4;

	4:(* Wait until read not busy *)
		fbFileGets( bExecute := FALSE, bError => bError, nErrID => nErrID, sLine => sCSVLine );
		IF NOT fbFileGets.bBusy THEN
			IF NOT fbFileGets.bError THEN
				IF fbFileGets.bEOF THEN
					step := 10;(* End of file reached => Close source file *)
				ELSE

					(* FB_FileGets returns text line without the CR (carriage return) character.
					We have to restore the CR character (replace the $L character with $R$L characters) *)
					IF RIGHT( sCSVLine, 1 ) = '$L' THEN
						sCSVLine := REPLACE( sCSVLine, '$R$L', 2, LEN( sCSVLine ) );
					END_IF

					step := 5;
				END_IF
			ELSE(* Error *)
				step := 100;
			END_IF
		END_IF

	5:(* Parse single line (record) *)
		fbReader.eCmd := eEnumCmd_First;(* Read first field value *)
		REPEAT
			fbReader( pBuffer := ADR( sCSVLine ), cbBuffer := SIZEOF( sCSVLine ), getValue => sCSVField );
			IF fbReader.bOk THEN
				fbReader.eCmd := eEnumCmd_Next;(* Read next field value *)

				IF ( nRow <= MAX_CSV_ROWS ) THEN
					IF ( nColumn <= MAX_CSV_COLUMNS ) THEN
						database[nRow, nColumn] := CSVFIELD_TO_STRING( sCSVField, FALSE );(* TODO: Save or use the field value in your application *)
					END_IF
				END_IF

				nColumn := nColumn + 1;(* Increment number of read columns *)
				IF fbReader.bCRLF THEN(* CRLF == TRUE => End of reacord reached *)
					nRow 		:= nRow + 1;(* Increment number of read records *)
					nColumn 	:= 0;(* Reset number of columns *)
				END_IF

			ELSE(* Error: End of record reached or all fields read *)
				step := 3;(* Try to read next line *)
			END_IF
		UNTIL NOT fbReader.bOk
		END_REPEAT

	10:	(* Close source file *)
		fbFileClose( bExecute := FALSE );
		fbFileClose( sNetId := sNetId, hFile := hFile, bExecute := TRUE );
		step := 11;

	11:(* Wait until close not busy *)
		fbFileClose( bExecute := FALSE, bError => bError, nErrID => nErrID );
		IF ( NOT fbFileClose.bBusy ) THEN
			hFile := 0;
			step := 100;
		END_IF

	100: (* Error or ready step => cleanup *)
		IF ( hFile <> 0 ) THEN
			step := 10; (* Close the source file *)
		ELSE
			bBusy := FALSE;
			step := 0;	(* Ready *)
		END_IF

END_CASE

END_PROGRAM

// ---- POUs/Item_Simulator/FBs/FB_ItemGenerator.TcPOU
FUNCTION_BLOCK FB_ItemGenerator
VAR_INPUT
	bStart				:BOOL;
	bStop				:BOOL;
	
	aStItemGen			:ARRAY[1..10] OF ST_ItemGenerator;
	stItemGenFromReg	:ST_ItemGenerator;
	
END_VAR
VAR
	//Item generators
	fbItemGen1			:FB_ClockPulsNumber;
	fbItemGen2			:FB_ClockPulsNumber;
	fbItemGen3			:FB_ClockPulsNumber;
	fbItemGen4			:FB_ClockPulsNumber;
	fbItemGen5			:FB_ClockPulsNumber;
	fbItemGen6			:FB_ClockPulsNumber;
	fbItemGen7			:FB_ClockPulsNumber;
	fbItemGen8			:FB_ClockPulsNumber;
	fbItemGen9			:FB_ClockPulsNumber;
	fbItemGen10			:FB_ClockPulsNumber;
	fbItemGenFromReg	:FB_ClockPulsNumber;
	
	//Sequence
	bInit				:BOOL := TRUE;
	eState				:E_ItemGenerator;
	
END_VAR

VAR_OUTPUT
	bSignalOutput		:BOOL;
END_VAR

//Init
IF bInit THEN
	eState := E_ItemGenerator.Idle;
	bInit := FALSE;
END_IF

//Call item generator cases
M_GeneratorCases();

//Reset Commands
bstart := FALSE;
bStop := FALSE;

METHOD PUBLIC M_GeneratorCases
VAR_INPUT
END_VAR

CASE eState OF
	
	// Idle
	E_ItemGenerator.Idle:
	
		// Reset generators
		fbItemGen1(
			bTrig := FALSE,
			bStop := TRUE,
			bPuls => bSignalOutput);
			
		fbItemGen2(
			bTrig := FALSE,
			bStop := TRUE,
			bPuls => bSignalOutput);
			
		fbItemGen3(
			bTrig := FALSE,
			bStop := TRUE,
			bPuls => bSignalOutput);
			
		fbItemGen4(
			bTrig := FALSE,
			bStop := TRUE,
			bPuls => bSignalOutput);
			
		fbItemGen5(
			bTrig := FALSE,
			bStop := TRUE,
			bPuls => bSignalOutput);
			
		fbItemGen6(
			bTrig := FALSE,
			bStop := TRUE,
			bPuls => bSignalOutput);
			
		fbItemGen7(
			bTrig := FALSE,
			bStop := TRUE,
			bPuls => bSignalOutput);
			
		fbItemGen8(
			bTrig := FALSE,
			bStop := TRUE,
			bPuls => bSignalOutput);
			
		fbItemGen9(
			bTrig := FALSE,
			bStop := TRUE,
			bPuls => bSignalOutput);
			
		fbItemGen10(
			bTrig := FALSE,
			bStop := TRUE,
			bPuls => bSignalOutput);
			
		fbItemGenFromReg(
			bTrig := FALSE,
			bStop := TRUE,
			bPuls => bSignalOutput);
	
		IF bStart THEN
			IF aStItemGen[1].bEnableGenerator THEN
				eState := E_ItemGenerator.ItemGenerator1;
			ELSE
				eState := E_ItemGenerator.ItemGeneratorFromRegistry;
			END_IF
		END_IF
		
		
		
	// Item generator 1
	E_ItemGenerator.ItemGenerator1:
	
		// If generator is enabled start the pulses
		IF NOT bStop THEN 

			fbItemGen1(
				bTrig			:= aStItemGen[1].bEnableGenerator, 
				bStop			:= FALSE,
				uiNo 			:= aStItemGen[1].nNumberOfPulses,  
				tPulsLengthOn 	:= aStItemGen[1].tTimeOnPulse,
				tPulsLengthOff 	:= aStItemGen[1].tTimeOffPulse,
				bPuls			=> bSignalOutput);
				
			// When all pulses have been made, go to generator 2
			IF fbItemGen1.uiCount >= (fbItemGen1.uiNo+1) THEN
				eState := E_ItemGenerator.ItemGenerator2;
			END_IF
			
		// If generator is not enabled, go to idle
		ELSE
			eState := E_ItemGenerator.Idle;
		END_IF;
		
		
		
	// Item generator 2
	E_ItemGenerator.ItemGenerator2:
	
		// If generator is enabled start the pulses
		IF aStItemGen[2].bEnableGenerator AND NOT bStop THEN 

			fbItemGen2(
				bTrig			:= aStItemGen[2].bEnableGenerator, 
				bStop			:= FALSE,
				uiNo 			:= aStItemGen[2].nNumberOfPulses, 
				tPulsLengthOn 	:= aStItemGen[2].tTimeOnPulse,
				tPulsLengthOff	:= aStItemGen[2].tTimeOffPulse,
				bPuls			=> bSignalOutput);
				
			// When all pulses have been made, go to generator 3
			IF fbItemGen2.uiCount >= (fbItemGen2.uiNo+1) THEN
				eState := E_ItemGenerator.ItemGenerator3;
			END_IF
			
		// If generator is not enabled, go to idle
		ELSE
			eState := E_ItemGenerator.Idle;
		END_IF;
		
		
		
		
	// Item generator 3
	E_ItemGenerator.ItemGenerator3:
	
		// If generator is enabled start the pulses
		IF astItemGen[3].bEnableGenerator AND NOT bStop THEN 

			fbItemGen3(
				bTrig			:= aStItemGen[3].bEnableGenerator, 
				bStop			:= FALSE,
				uiNo 			:= aStItemGen[3].nNumberOfPulses, 
				tPulsLengthOn 	:= aStItemGen[3].tTimeOnPulse,
				tPulsLengthOff 	:= aStItemGen[3].tTimeOffPulse,
				bPuls			=> bSignalOutput);
				
			// When all pulses have been made, go to generator 4
			IF fbItemGen3.uiCount >= (fbItemGen3.uiNo+1) THEN
				eState := E_ItemGenerator.ItemGenerator4;
			END_IF
			
		// If generator is not enabled, go to idle
		ELSE
			eState := E_ItemGenerator.Idle;
		END_IF;
		
		
	// Item generator 4
	E_ItemGenerator.ItemGenerator4:
	
		// If generator is enabled start the pulses
		IF aStItemGen[4].bEnableGenerator AND NOT bStop THEN 

			fbItemGen4(
				bTrig			:= aStItemGen[4].bEnableGenerator, 
				bStop			:= FALSE,
				uiNo 			:= aStItemGen[4].nNumberOfPulses, 
				tPulsLengthOn 	:= aStItemGen[4].tTimeOnPulse,
				tPulsLengthOff 	:= aStItemGen[4].tTimeOffPulse,
				bPuls			=> bSignalOutput);
				
			// When all pulses have been made, go to generator 5
			IF fbItemGen4.uiCount >= (fbItemGen4.uiNo+1) THEN
				eState := E_ItemGenerator.ItemGenerator5;
			END_IF
			
		// If generator is not enabled, go to idle
		ELSE
			eState := E_ItemGenerator.Idle;
		END_IF;
		
		
	// Item generator 5
	E_ItemGenerator.ItemGenerator5:
	
		// If generator is enabled start the pulses
		IF aStItemGen[5].bEnableGenerator AND NOT bStop THEN 

			fbItemGen5(
				bTrig			:= aStItemGen[5].bEnableGenerator, 
				bStop			:= FALSE,
				uiNo 			:= aStItemGen[5].nNumberOfPulses, 
				tPulsLengthOn 	:= aStItemGen[5].tTimeOnPulse,
				tPulsLengthOff 	:= aStItemGen[5].tTimeOffPulse,
				bPuls			=> bSignalOutput);
				
			// When all pulses have been made, go to generator 6
			IF fbItemGen5.uiCount >= (fbItemGen5.uiNo+1) THEN
				eState := E_ItemGenerator.ItemGenerator6;
			END_IF
			
		// If generator is not enabled, go to idle
		ELSE
			eState := E_ItemGenerator.Idle;
		END_IF;
		
	
	// Item generator 6
	E_ItemGenerator.ItemGenerator6:
	
		// If generator is enabled start the pulses
		IF aStItemGen[6].bEnableGenerator AND NOT bStop THEN 

			fbItemGen6(
				bTrig			:= aStItemGen[6].bEnableGenerator, 
				bStop			:= FALSE,
				uiNo 			:= aStItemGen[6].nNumberOfPulses, 
				tPulsLengthOn 	:= aStItemGen[6].tTimeOnPulse,
				tPulsLengthOff 	:= aStItemGen[6].tTimeOffPulse,
				bPuls			=> bSignalOutput);
				
			// When all pulses have been made, go to generator 7
			IF fbItemGen6.uiCount >= (fbItemGen6.uiNo+1) THEN
				eState := E_ItemGenerator.ItemGenerator7;
			END_IF
			
		// If generator is not enabled, go to idle
		ELSE
			eState := E_ItemGenerator.Idle;
		END_IF;
		
		
	// Item generator 7
	E_ItemGenerator.ItemGenerator7:
	
		// If generator is enabled start the pulses
		IF aStItemGen[7].bEnableGenerator AND NOT bStop THEN 

			fbItemGen7(
				bTrig			:= aStItemGen[7].bEnableGenerator, 
				bStop			:= FALSE,
				uiNo 			:= aStItemGen[7].nNumberOfPulses, 
				tPulsLengthOn 	:= aStItemGen[7].tTimeOnPulse,
				tPulsLengthOff 	:= aStItemGen[7].tTimeOffPulse,
				bPuls			=> bSignalOutput);
				
			// When all pulses have been made, go to generator 8
			IF fbItemGen7.uiCount >= (fbItemGen7.uiNo+1) THEN
				eState := E_ItemGenerator.ItemGenerator8;
			END_IF
			
		// If generator is not enabled, go to idle
		ELSE
			eState := E_ItemGenerator.Idle;
		END_IF;
		
		
	// Item generator 8
	E_ItemGenerator.ItemGenerator8:
	
		// If generator is enabled start the pulses
		IF aStItemGen[8].bEnableGenerator AND NOT bStop THEN 

			fbItemGen8(
				bTrig			:= aStItemGen[8].bEnableGenerator, 
				bStop			:= FALSE,
				uiNo 			:= aStItemGen[8].nNumberOfPulses, 
				tPulsLengthOn 	:= aStItemGen[8].tTimeOnPulse,
				tPulsLengthOff 	:= aStItemGen[8].tTimeOffPulse,
				bPuls			=> bSignalOutput);
				
			// When all pulses have been made, go to generator 9
			IF fbItemGen8.uiCount >= (fbItemGen8.uiNo+1) THEN
				eState := E_ItemGenerator.ItemGenerator9;
			END_IF
			
		// If generator is not enabled, go to idle
		ELSE
			eState := E_ItemGenerator.Idle;
		END_IF;
		
		
	// Item generator 9
	E_ItemGenerator.ItemGenerator9:
	
		// If generator is enabled start the pulses
		IF aStItemGen[9].bEnableGenerator AND NOT bStop THEN 

			fbItemGen9(
				bTrig			:= aStItemGen[9].bEnableGenerator, 
				bStop			:= FALSE,
				uiNo 			:= aStItemGen[9].nNumberOfPulses, 
				tPulsLengthOn 	:= aStItemGen[9].tTimeOnPulse,
				tPulsLengthOff 	:= aStItemGen[9].tTimeOffPulse, 
				bPuls			=> bSignalOutput);
				
			// When all pulses have been made, go to generator 10
			IF fbItemGen9.uiCount >= (fbItemGen9.uiNo+1) THEN
				eState := E_ItemGenerator.ItemGenerator10;
			END_IF
			
		// If generator is not enabled, go to idle
		ELSE
			eState := E_ItemGenerator.Idle;
		END_IF;
		
		
	// Item generator 10
	E_ItemGenerator.ItemGenerator10:
	
		// If generator is enabled start the pulses
		IF aStItemGen[10].bEnableGenerator AND NOT bStop THEN 

			fbItemGen10(
				bTrig			:= aStItemGen[10].bEnableGenerator, 
				bStop			:= FALSE,
				uiNo 			:= aStItemGen[10].nNumberOfPulses, 
				tPulsLengthOn 	:= aStItemGen[10].tTimeOnPulse,
				tPulsLengthOff 	:= aStItemGen[10].tTimeOffPulse, 
				bPuls			=> bSignalOutput);
				
			// When all pulses have been made, go to Idle
			IF fbItemGen10.uiCount >= (fbItemGen10.uiNo+1) THEN
				eState := E_ItemGenerator.Idle;
			END_IF
			
		// If generator is not enabled, go to idle
		ELSE
			eState := E_ItemGenerator.Idle;
		END_IF;
		
		
	// Item generator from registry
	E_ItemGenerator.ItemGeneratorFromRegistry:
	
		// If generator is enabled start the pulses
		IF stItemGenFromReg.bEnableGenerator AND NOT bStop THEN 

			fbItemGenFromReg(
				bTrig			:= stItemGenFromReg.bEnableGenerator, 
				bStop			:= FALSE,
				uiNo 			:= stItemGenFromReg.nNumberOfPulses, 
				tPulsLengthOn 	:= stItemGenFromReg.tTimeOnPulse,
				tPulsLengthOff 	:= stItemGenFromReg.tTimeOffPulse, 
				bPuls			=> bSignalOutput);
				
			// When all pulses have been made, go to Idle
			IF fbItemGenFromReg.uiCount >= (fbItemGenFromReg.uiNo+1) THEN
				eState := E_ItemGenerator.Idle;
			END_IF
			
		// If generator is not enabled, go to idle
		ELSE
			eState := E_ItemGenerator.Idle;
		END_IF;
		
END_CASE
END_METHOD

END_FUNCTION_BLOCK

// ---- POUs/Item_Simulator/FBs/FB_ItemRegister.TcPOU
FUNCTION_BLOCK FB_ItemRegister
VAR_INPUT
	bSignal					: BOOL;
	bReset					: BOOL;
END_VAR
VAR_OUTPUT
	aItemOnTimeRegistry		: ARRAY[0..GVL_Constant.ITEM_ARRAY_SIZE] OF TIME;
	aItemOffTimeRegistry	: ARRAY[0..GVL_Constant.ITEM_ARRAY_SIZE] OF TIME;
	
	nTimeCount				: INT;
END_VAR
VAR
	tTimeOn					: TON;
	tReadTimeOn				: TIME;
	osReadOnTime			: F_TRIG;
	
	tTimeOFF				: TON;
	tReadTimeOff			: TIME;
	osReadOffTime			: R_TRIG;
	
	i						: INT;
END_VAR

IF bSignal THEN
	tTimeOn(IN:=TRUE, PT:=T#5S, ET=>tReadTimeOn);
ELSE
	tTimeOFF(IN:=TRUE, PT:=T#5S, ET=>tReadTimeOff);
END_IF;

//Write on time to array
A_ReadOnTime();

//Write off time to array
A_ReadOffTime();

//Reset array for time registry
A_ResetTimeRegistry();

ACTION A_ReadOffTime:
osReadOffTime(CLK:=bSignal);

IF osReadOffTime.Q THEN
	aItemOffTimeRegistry[nTimeCount] := tReadTimeOff;
	tTimeOff(IN:=FALSE);
END_IF
END_ACTION

ACTION A_ReadOnTime:
osReadOnTime(CLK:=bSignal);

IF osReadOnTime.Q THEN
	aItemOnTimeRegistry[nTimeCount] := tReadTimeOn;
	nTimeCount := nTimeCount +1;
	tTimeOn(IN:=FALSE);
END_IF
END_ACTION

ACTION A_ResetTimeRegistry:
IF bReset THEN
	tTimeOFF(IN:=FALSE);
	tTimeOn(IN:=FALSE);
	
	FOR i := 0 TO nTimeCount DO 
		aItemOffTimeRegistry[i] := T#0S;
		aItemOnTimeRegistry [i] := T#0S;
	END_FOR
	
	nTimeCount := 0;	
	bReset := FALSE;
END_IF
END_ACTION

END_FUNCTION_BLOCK

// ---- GlobalTextList.TcGTLO
TEXTLIST GlobalTextList
  588 = '!! Generator from registry must not be enabled while other generators are enabled. !!'
  942 = '%i'
  636 = '%s'
  153 = 'ADS return code: %i'
  144 = 'ADS Status: %s'
  701 = 'aItemOnTimeRegistry[INDEX]'
  930 = 'Camera Output Timestamp'
  148 = 'Camera Port Timestamp'
  690 = 'Delta Time In MS'
  156 = 'Delta Time in MS'
  531 = 'Delta Time MS'
  96 = 'Digital Input Timestamp'
  739 = 'Digital Output Timestamo'
  466 = 'Digital Output Timestamp'
  81 = 'Digital Sensor Timestamp'
  490 = 'EAN From Registry'
  146 = 'EAN String From Registry'
  668 = 'Enable Generator 1'
  296 = 'Enable Generator 10'
  294 = 'Enable Generator 2'
  902 = 'Enable Generator 3'
  752 = 'Enable Generator 4'
  927 = 'Enable Generator 5'
  28 = 'Enable Generator 6'
  464 = 'Enable Generator 7'
  726 = 'Enable Generator 8'
  800 = 'Enable Generator 9'
  459 = 'Enable Generator From Registry'
  141 = 'Enabled'
  143 = 'Error step: %s'
  147 = 'Errors : %i'
  826 = 'Export CSV File'
  834 = 'Generator from registry must not be enabled while other generators are enabled.'
  578 = 'Import CSV File'
  152 = 'Init'
  551 = 'Item Generator'
  155 = 'Items generated'
  150 = 'LinkOk'
  442 = 'Number of items'
  129 = 'Off time'
  423 = 'Off time From Registry'
  963 = 'Off Time From Registry'
  657 = 'On time'
  878 = 'On time From Registry'
  784 = 'PC Port Timestamp'
  479 = 'PRG_Simulator.stItemGen1.nNumberOfPulses'
  465 = 'Read CSV'
  207 = 'Read From Camera TCP'
  628 = 'Read From PC TCP'
  95 = 'Read From TCP'
  145 = 'Reads : %i'
  151 = 'Remote NetId: %s'
  847 = 'Reset Registry'
  33 = 'Sesnor Input Timestamp'
  271 = 'Start Generator'
  828 = 'Start Generator Sequence'
  140 = 'Step: %s'
  971 = 'Stop Generator'
  684 = 'Stop Generator Sequence'
  97 = 'TCP Camera Timestamp'
  13 = 'TCP Port Timestamp'
  154 = 'Time e. : %i'
  928 = 'View Simulator'
  24 = 'View Timestamps'
  102 = 'Write CSV'
  383 = 'Write To Camera TCP'
  365 = 'Write To TCP'
END_TEXTLIST

// ---- POUs/00_BuildingBlocks/PlcToPlcCom/DUTs/ADS_ErrorCodes.TcTLO
TEXTLIST ADS_ErrorCodes
  1 = 'Internal error'
  6 = 'target port not found. ADS Server not started '
  7 = 'target machine not found. Missing ADS routes '
  13 = 'Port not connected'
  14 = 'Invalid ADS length'
  15 = 'Invalid ADS Net ID'
  18 = 'Port disabled'
  19 = 'Port already connected'
  24 = 'Invalid ADS port'
  26 = 'TCP send error'
  27 = 'Host unreachable'
  28 = 'Invalid AMS fragment'
  1792 = 'error class <device error> '
  1793 = 'Service is not supported by server   '
  1794 = 'invalid index group  '
  1795 = 'invalid index offset    '
  1796 = 'reading/writing not permitted     '
  1797 = 'parameter size not correct'
  1798 = 'invalid parameter value(s)     '
  1799 = 'device is not in a ready state'
  1800 = 'device is busy '
  1801 = 'invalid context (must be in Windows) '
  1802 = 'out of memory '
  1803 = 'invalid parameter value(s)'
  1804 = 'not found (files, ...) '
  1805 = 'syntax error in command or file   '
  1806 = 'objects do not match '
  1807 = 'object already exists '
  1808 = 'symbol not found '
  1809 = 'symbol version invalid Onlinechange Release handle and get a new one '
  1810 = 'server is in invalid state'
  1811 = 'AdsTransMode not supported '
  1812 = 'Notification handle is invalid Onlinechange Release handle and get a new one '
  1813 = 'Notification client not registered  '
  1814 = 'no more notification handles'
  1815 = 'size for watch too big  '
  1816 = 'device not initialized'
  1817 = 'device has a timeout '
  1818 = 'query interface failed'
  1819 = 'wrong interface required'
  1820 = 'class ID is invalid'
  1821 = 'object ID is invalid'
  1822 = 'request is pending  '
  1823 = 'request is aborted'
  1824 = 'signal warning'
  1825 = 'invalid array index   '
  1826 = 'symbol not active Onlinechange Release handle and get a new one '
  1827 = 'access denied  '
  1828 = 'missing license   Activate license for TwinCAT 3 function '
  1836 = 'exception occured during system start  Check each device transistions'
  1856 = 'Error class client error '
  1857 = 'invalid parameter at service '
  1858 = 'polling list is empty'
  1859 = 'var connection already in use '
  1860 = 'invoke ID in use  '
  1861 = 'timeout elapsed   Check ADS routes of sender and receiver and your  firewall setting'
  1862 = 'error in win32 subsystem'
  1863 = 'Invalid client timeout value '
  1864 = 'ads-port not opened'
  1872 = 'internal error in ads sync'
  1873 = 'hash table overflow '
  1874 = 'key not found in hash'
  1875 = 'no more symbols in cache'
  1876 = 'invalid response received'
  1877 = 'sync port is locked'
  0 = 'no error'
   = 'See ADS returncode at the manual'
   = ''
END_TEXTLIST

// ---- POUs/00_BuildingBlocks/PlcToPlcCom/VIZU_PlcAdsRead.TcVIS
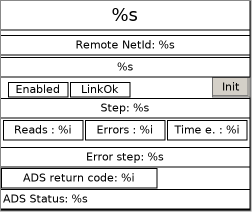
VISUALIZATION VIZU_PlcAdsRead  // 252x212
VAR_INPUT
	sName : STRING; 
END_VAR
VAR_IN_OUT
	stHmi : ST_PlcAdsReadHmi; //Hmi data
END_VAR
    Rectangle (0,0 250x210)
    Rectangle (0,0 250x30), "%s", text variable: sName
    Rectangle (0,98 250x20), "Step: %s", text variable: stHmi.eS_Step
    Rectangle (8,82 60x15), "Enabled", colour toggle: stHmi.bS_Enable
    Rectangle (0,147 250x20), "Error step: %s", text variable: stHmi.eS_ErrorStep, colour toggle: stHmi.bS_Error
    Rectangle (0,189 250x20), "ADS Status: %s", text list: 'ADS_ErrorCodes', text index: stHmi.udiS_ErrorId
    Rectangle (3,120 80x20), "Reads : %i", text variable: stHmi.udiS_ReadCount
        OnMouseClick: write the text variable via Default
    Rectangle (85,120 80x20), "Errors : %i", text variable: stHmi.udiS_ReadErrors
        OnMouseClick: write the text variable via Default
    Rectangle (70,82 60x15), "LinkOk", colour toggle: stHmi.bS_LinkOk
    Rectangle (0,35 250x20), "Remote NetId: %s", text variable: stHmi.sRemoteId
    Button (212,77 38x20), "Init"
        tap stHmi.bC_Init
    Rectangle (0,57 250x20), "%s", text variable: stHmi.sRemoteSymbol
    Rectangle (1,168 156x20), "ADS return code: %i", text variable: stHmi.udiS_ErrorId
    Rectangle (167,120 80x20), "Time e. : %i", text variable: stHmi.udiS_ReadIntervalErrors
        OnMouseClick: write the text variable via Default
END_VISUALIZATION

// ---- VISUs/ItemSimulator.TcVIS
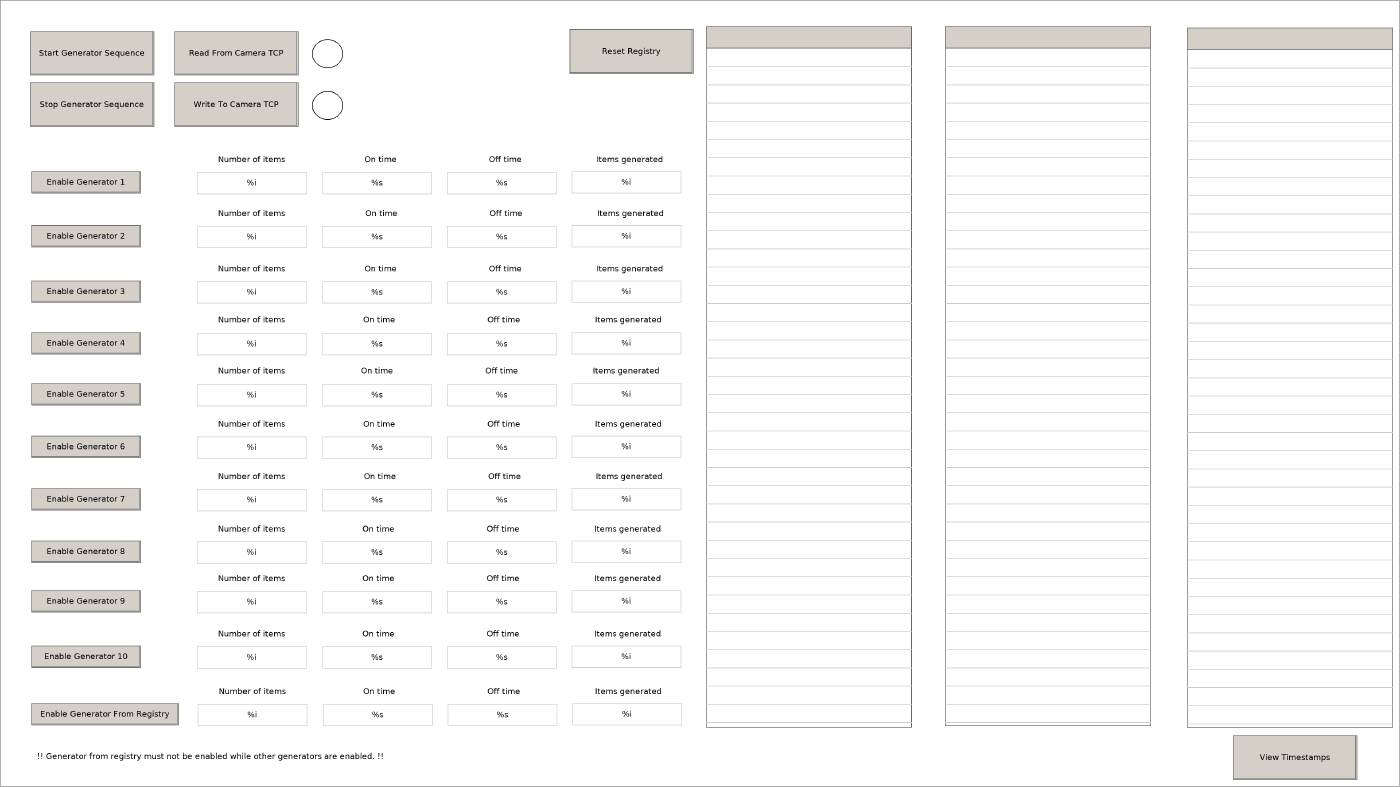
VISUALIZATION ItemSimulator  // 1920x1080
    Button (43,235 150x30), "Enable Generator 1", colour toggle: PRG_Simulator.stItemGen1.bEnableGenerator
        toggle PRG_Simulator.fbItemGenerator.aStItemGen[1].bEnableGenerator
    Textfield (270,236 150x30), "%i", text variable: PRG_Simulator.stItemGen1.nNumberOfPulses
        OnMouseClick: write the text variable via Default
    Textfield (442,236 150x30), "%s", text variable: PRG_Simulator.stItemGen1.tTimeOnPulse, text index: PRG_Simulator.stItemGen1.tTimeOnPulse
        OnMouseClick: write the text variable via Default
    Textfield (613,236 150x30), "%s", text variable: PRG_Simulator.stItemGen1.tTimeOffPulse, text index: PRG_Simulator.stItemGen1.tTimeOffPulse
        OnMouseClick: write the text variable via Default
    Label (270,204 150x30), "Number of items"
    Label (447,204 150x30), "On time"
    Label (618,204 150x30), "Off time"
    Textfield (784,235 150x30), "%i", text variable: PRG_Simulator.fbItemGenerator.fbItemGen1.uiCount, input disabled if: TRUE, text index: PRG_Simulator.stItemGen1.nNumberOfPulses
        OnMouseClick: write the text variable via Default
    Label (789,204 150x30), "Items generated"
    Button (41,43 170x60), "Start Generator Sequence"
        OnMouseDown: execute { GVL_HMI.stItemSimulator.bStartGenerator := TRUE; }
    Button (41,113 170x61), "Stop Generator Sequence"
        OnMouseDown: execute { GVL_HMI.stItemSimulator.bStopGenerator := TRUE; }
    Button (43,309 150x30), "Enable Generator 2", colour toggle: PRG_Simulator.stItemGen2.bEnableGenerator
        toggle PRG_Simulator.fbItemGenerator.aStItemGen[2].bEnableGenerator
    Textfield (270,310 150x30), "%i", text variable: PRG_Simulator.stItemGen2.nNumberOfPulses
        OnMouseClick: write the text variable via Default
    Textfield (442,310 150x30), "%s", text variable: PRG_Simulator.stItemGen2.tTimeOnPulse
        OnMouseClick: write the text variable via Default
    Textfield (613,310 150x30), "%s", text variable: PRG_Simulator.stItemGen2.tTimeOffPulse
        OnMouseClick: write the text variable via Default
    Label (270,278 150x30), "Number of items"
    Label (448,278 150x30), "On time"
    Label (619,278 150x30), "Off time"
    Textfield (784,309 150x30), "%i", text variable: PRG_Simulator.fbItemGenerator.fbItemGen2.uiCount, input disabled if: TRUE
        OnMouseClick: write the text variable via Default
    Label (790,278 150x30), "Items generated"
    Button (43,385 150x30), "Enable Generator 3", colour toggle: PRG_Simulator.stItemGen3.bEnableGenerator
        toggle PRG_Simulator.fbItemGenerator.aStItemGen[3].bEnableGenerator
    Textfield (270,386 150x30), "%i", text variable: PRG_Simulator.stItemGen3.nNumberOfPulses
        OnMouseClick: write the text variable via Default
    Textfield (442,386 150x30), "%s", text variable: PRG_Simulator.stItemGen3.tTimeOnPulse
        OnMouseClick: write the text variable via Default
    Textfield (613,386 150x30), "%s", text variable: PRG_Simulator.stItemGen3.tTimeOffPulse
        OnMouseClick: write the text variable via Default
    Label (270,354 150x30), "Number of items"
    Label (447,354 150x30), "On time"
    Label (618,354 150x30), "Off time"
    Textfield (784,385 150x30), "%i", text variable: PRG_Simulator.fbItemGenerator.fbItemGen3.uiCount, input disabled if: TRUE
        OnMouseClick: write the text variable via Default
    Label (789,354 150x30), "Items generated"
    Button (43,456 150x30), "Enable Generator 4", colour toggle: PRG_Simulator.stItemGen4.bEnableGenerator
        toggle PRG_Simulator.fbItemGenerator.aStItemGen[4].bEnableGenerator
    Textfield (270,457 150x30), "%i", text variable: PRG_Simulator.stItemGen4.nNumberOfPulses
        OnMouseClick: write the text variable via Default
    Textfield (442,457 150x30), "%s", text variable: PRG_Simulator.stItemGen4.tTimeOnPulse
        OnMouseClick: write the text variable via Default
    Textfield (613,457 150x30), "%s", text variable: PRG_Simulator.stItemGen4.tTimeOffPulse
        OnMouseClick: write the text variable via Default
    Label (270,424 150x30), "Number of items"
    Label (445,424 150x30), "On time"
    Label (616,424 150x30), "Off time"
    Textfield (784,456 150x30), "%i", text variable: PRG_Simulator.fbItemGenerator.fbItemGen4.uiCount, input disabled if: TRUE
        OnMouseClick: write the text variable via Default
    Label (787,424 150x30), "Items generated"
    Button (43,526 150x30), "Enable Generator 5", colour toggle: PRG_Simulator.stItemGen5.bEnableGenerator
        toggle PRG_Simulator.fbItemGenerator.aStItemGen[5].bEnableGenerator
    Textfield (270,527 150x30), "%i", text variable: PRG_Simulator.stItemGen5.nNumberOfPulses
        OnMouseClick: write the text variable via Default
    Textfield (442,527 150x30), "%s", text variable: PRG_Simulator.stItemGen5.tTimeOnPulse
        OnMouseClick: write the text variable via Default
    Textfield (613,527 150x30), "%s", text variable: PRG_Simulator.stItemGen5.tTimeOffPulse
        OnMouseClick: write the text variable via Default
    Label (270,494 150x30), "Number of items"
    Label (442,494 150x30), "On time"
    Label (613,494 150x30), "Off time"
    Textfield (784,526 150x30), "%i", text variable: PRG_Simulator.fbItemGenerator.fbItemGen5.uiCount, input disabled if: TRUE
        OnMouseClick: write the text variable via Default
    Label (784,494 150x30), "Items generated"
    Button (43,598 150x30), "Enable Generator 6", colour toggle: PRG_Simulator.stItemGen6.bEnableGenerator
        toggle PRG_Simulator.fbItemGenerator.aStItemGen[6].bEnableGenerator
    Textfield (270,599 150x30), "%i", text variable: PRG_Simulator.stItemGen6.nNumberOfPulses
        OnMouseClick: write the text variable via Default
    Textfield (442,599 150x30), "%s", text variable: PRG_Simulator.stItemGen6.tTimeOnPulse
        OnMouseClick: write the text variable via Default
    Textfield (613,599 150x30), "%s", text variable: PRG_Simulator.stItemGen6.tTimeOffPulse
        OnMouseClick: write the text variable via Default
    Label (270,567 150x30), "Number of items"
    Label (445,567 150x30), "On time"
    Label (616,567 150x30), "Off time"
    Textfield (784,598 150x30), "%i", text variable: PRG_Simulator.fbItemGenerator.fbItemGen6.uiCount, input disabled if: TRUE
        OnMouseClick: write the text variable via Default
    Label (787,567 150x30), "Items generated"
    Button (43,670 150x30), "Enable Generator 7", colour toggle: PRG_Simulator.stItemGen7.bEnableGenerator
        toggle PRG_Simulator.fbItemGenerator.aStItemGen[7].bEnableGenerator
    Textfield (270,671 150x30), "%i", text variable: PRG_Simulator.stItemGen7.nNumberOfPulses
        OnMouseClick: write the text variable via Default
    Textfield (442,671 150x30), "%s", text variable: PRG_Simulator.stItemGen7.tTimeOnPulse
        OnMouseClick: write the text variable via Default
    Textfield (613,671 150x30), "%s", text variable: PRG_Simulator.stItemGen7.tTimeOffPulse
        OnMouseClick: write the text variable via Default
    Label (270,639 150x30), "Number of items"
    Label (446,639 150x30), "On time"
    Label (617,639 150x30), "Off time"
    Textfield (784,670 150x30), "%i", text variable: PRG_Simulator.fbItemGenerator.fbItemGen7.uiCount, input disabled if: TRUE
        OnMouseClick: write the text variable via Default
    Label (788,639 150x30), "Items generated"
    Button (43,742 150x30), "Enable Generator 8", colour toggle: PRG_Simulator.stItemGen8.bEnableGenerator
        toggle PRG_Simulator.fbItemGenerator.aStItemGen[8].bEnableGenerator
    Textfield (270,743 150x30), "%i", text variable: PRG_Simulator.stItemGen8.nNumberOfPulses
        OnMouseClick: write the text variable via Default
    Textfield (442,743 150x30), "%s", text variable: PRG_Simulator.stItemGen8.tTimeOnPulse
        OnMouseClick: write the text variable via Default
    Textfield (613,743 150x30), "%s", text variable: PRG_Simulator.stItemGen8.tTimeOffPulse
        OnMouseClick: write the text variable via Default
    Label (270,711 150x30), "Number of items"
    Label (444,711 150x30), "On time"
    Label (615,711 150x30), "Off time"
    Textfield (784,742 150x30), "%i", text variable: PRG_Simulator.fbItemGenerator.fbItemGen8.uiCount, input disabled if: TRUE
        OnMouseClick: write the text variable via Default
    Label (786,711 150x30), "Items generated"
    Button (43,810 150x30), "Enable Generator 9", colour toggle: PRG_Simulator.stItemGen9.bEnableGenerator
        toggle PRG_Simulator.fbItemGenerator.aStItemGen[9].bEnableGenerator
    Textfield (270,811 150x30), "%i", text variable: PRG_Simulator.stItemGen9.nNumberOfPulses
        OnMouseClick: write the text variable via Default
    Textfield (442,811 150x30), "%s", text variable: PRG_Simulator.stItemGen9.tTimeOnPulse
        OnMouseClick: write the text variable via Default
    Textfield (613,811 150x30), "%s", text variable: PRG_Simulator.stItemGen9.tTimeOffPulse
        OnMouseClick: write the text variable via Default
    Label (270,779 150x30), "Number of items"
    Label (444,779 150x30), "On time"
    Label (615,779 150x30), "Off time"
    Textfield (784,810 150x30), "%i", text variable: PRG_Simulator.fbItemGenerator.fbItemGen9.uiCount, input disabled if: TRUE
        OnMouseClick: write the text variable via Default
    Label (786,779 150x30), "Items generated"
    Button (43,886 150x30), "Enable Generator 10", colour toggle: PRG_Simulator.stItemGen10.bEnableGenerator
        toggle PRG_Simulator.fbItemGenerator.aStItemGen[10].bEnableGenerator
    Textfield (270,887 150x30), "%i", text variable: PRG_Simulator.stItemGen10.nNumberOfPulses
        OnMouseClick: write the text variable via Default
    Textfield (442,887 150x30), "%s", text variable: PRG_Simulator.stItemGen10.tTimeOnPulse
        OnMouseClick: write the text variable via Default
    Textfield (613,887 150x30), "%s", text variable: PRG_Simulator.stItemGen10.tTimeOffPulse
        OnMouseClick: write the text variable via Default
    Label (270,855 150x30), "Number of items"
    Label (444,855 150x30), "On time"
    Label (615,855 150x30), "Off time"
    Textfield (784,886 150x30), "%i", text variable: PRG_Simulator.fbItemGenerator.fbItemGen10.uiCount, input disabled if: TRUE
        OnMouseClick: write the text variable via Default
    Label (786,855 150x30), "Items generated"
    Textfield (271,966 150x30), "%i", text variable: PRG_Simulator.stItemGenFromReg.nNumberOfPulses, input disabled if: TRUE
        OnMouseClick: write the text variable via Default
    Textfield (443,966 150x30), "%s", text variable: PRG_Simulator.stItemGenFromReg.tTimeOnPulse, input disabled if: TRUE
        OnMouseClick: write the text variable via Default
    Textfield (614,966 150x30), "%s", text variable: PRG_Simulator.stItemGenFromReg.tTimeOffPulse, input disabled if: TRUE
        OnMouseClick: write the text variable via Default
    Label (271,934 150x30), "Number of items"
    Label (445,934 150x30), "On time"
    Label (616,934 150x30), "Off time"
    Textfield (785,965 150x30), "%i", text variable: PRG_Simulator.fbItemGenerator.fbItemGenFromReg.uiCount, input disabled if: TRUE
        OnMouseClick: write the text variable via Default
    Label (787,934 150x30), "Items generated"
    Button (43,965 202x30), "Enable Generator From Registry", colour toggle: PRG_Simulator.stItemGenFromReg.bEnableGenerator
        toggle PRG_Simulator.fbItemGenerator.stItemGenFromReg.bEnableGenerator
    Table (968,36 282x962), data array: PRG_Simulator.aItemOnTimeRegistry
        p3854506369: PRG_Simulator.aItemOnTimeRegistry[INDEX]
        p2232123230: On time From Registry
    Table (1296,36 282x960), data array: PRG_Simulator.aItemOffTimeRegistry
        p3854506369: PRG_Simulator.aItemOffTimeRegistry[INDEX]
        p2232123230: Off Time From Registry
    Button (781,40 170x61), "Reset Registry"
        OnMouseDown: execute { GVL_HMI.stItemSimulator.bResetRegistry := TRUE; GVL_HMI.stTCPConnection.bResetRegistry := TRUE; }
    Label (20,1023 537x30), "!! Generator from registry must not be enabled while other generators are enabled. !!"
    Table (1628,38 282x960), data array: GVL_HMI.stTCPConnectionStatus.aEANRegistry
        p3854506369: GVL_HMI.stTCPConnectionStatus.aEANRegistry[INDEX]
        p2232123230: EAN From Registry
    Button (239,43 170x60), "Read From Camera TCP"
        OnMouseDown: execute { GVL_HMI.stTCPConnectionCmd.bReadSocketConnect := TRUE; }
    Button (239,113 170x61), "Write To Camera TCP"
        OnMouseDown: execute { GVL_HMI.stTCPConnectionCmd.bWriteSocketConnect := TRUE; }
    Button (1691,1009 170x61), "View Timestamps"
        OnMouseClick: change screen: TimeStampOnItems
    Ellipse (428,54 42x39), colour toggle: GVL_HMI.stTCPConnectionStatus.bCameraReadSocketIsConnected, colour variable: 16#FFFFFFFF
        p2167032090: 16#FF78CE22
    Ellipse (428,125 42x39), colour toggle: GVL_HMI.stTCPConnectionStatus.bHlzWriteSocketIsConnected, colour variable: 16#FFFFFFFF
        p2167032090: 16#FF78CE22
END_VISUALIZATION

// ---- VISUs/TimeStampOnItems.TcVIS
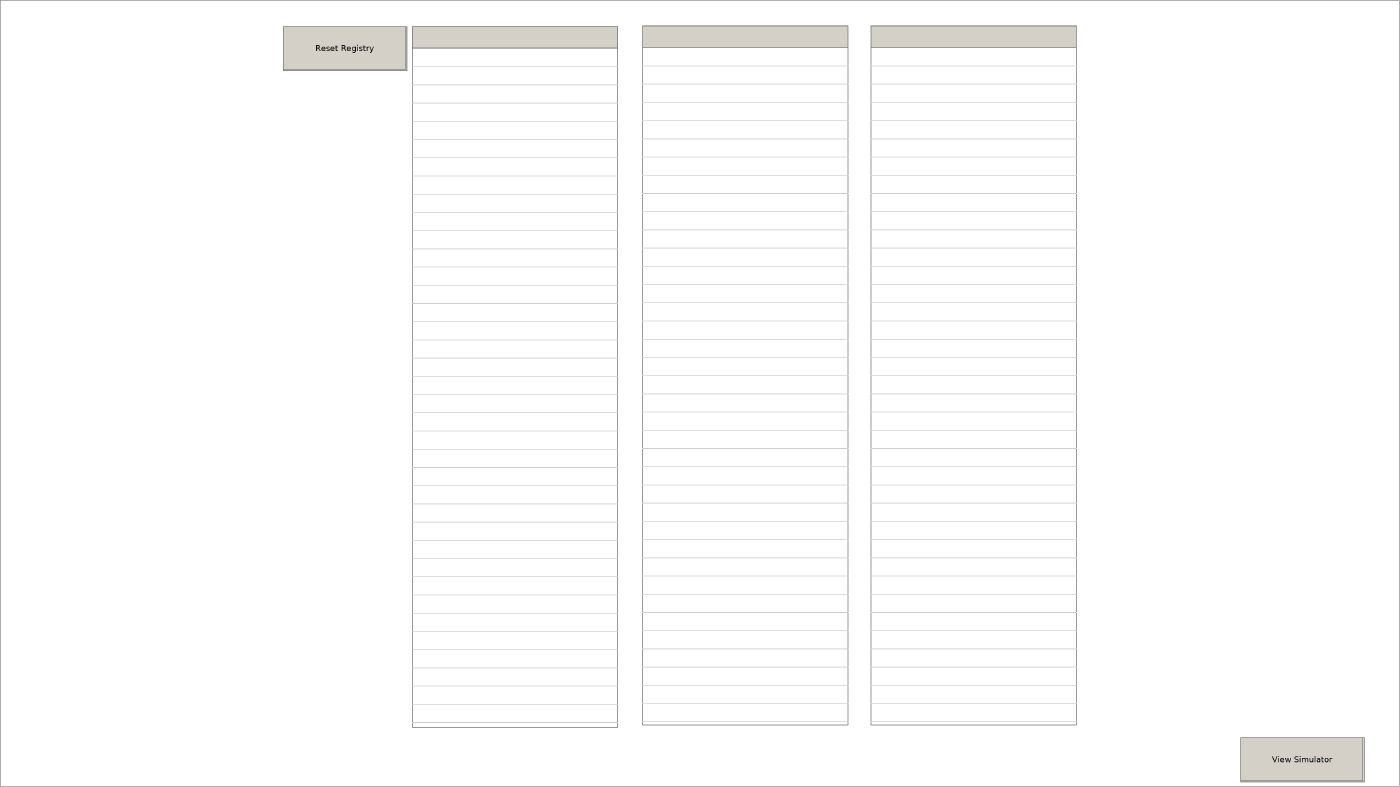
VISUALIZATION TimeStampOnItems  // 1920x1080
    Table (565,36 282x962), data array: GVL_HMI.stTimestampStatus.aDigitalSensorTime
        p3854506369: GVL_HMI.stTimestampStatus.aDigitalSensorTime[INDEX]
        p2232123230: Digital Sensor Timestamp
    Table (881,35 282x960), data array: GVL_HMI.stTimestampStatus.aTCPPortCameraTime
        p3854506369: GVL_HMI.stTimestampStatus.aTCPPortCameraTime[INDEX]
        p2232123230: TCP Camera Timestamp
    Button (388,36 170x61), "Reset Registry"
        OnMouseDown: execute { GVL_HMI.stTimestampCmd.bResetRegistry := TRUE; }
    Button (1701,1012 170x61), "View Simulator"
        OnMouseClick: change screen: ItemSimulator
    Table (1194,35 282x960), data array: GVL_HMI.stTimestampStatus.aDeltaTimeMS
        p3854506369: GVL_HMI.stTimestampStatus.aDeltaTimeMS[INDEX]
        p2232123230: Delta Time in MS
END_VISUALIZATION
